BEGIN
	//=============================================================================
	// SIEMENS AG
	// (c)Copyright 2023
	//-----------------------------------------------------------------------------
	// Library:       LKinCtrl
	// Tested with:   S7-1518TF-4 PN/DP, FW V3.1
	// Engineering:   TIA Portal V19
	// Restrictions:  ---
	// Requirements:  S7-1500T, FW V3.0
	// Functionality: Calc rotation axis and angle from rotation matrix
	// Support: tech.team.motioncontrol@siemens.com
	// Note: Parameter comments are only available in language 'English (United States)'
	//-----------------------------------------------------------------------------
	// Change log table:
	// Version  Date       Expert in charge Changes applied
	// 01.00.00 21.09.2023 SF               First released version
	//=============================================================================
	
	#tempRadDeg := 180.0 / #PI;
	#tempRotAngle := ACOS((#rotMatrix[1, 1] + #rotMatrix[2, 2] + #rotMatrix[3, 3] - 1.0) * 0.5);
	
	IF (#tempRotAngle = 0.0) THEN
	  // No rotation
	  #tempR1 := 0.0;
	  #tempR2 := 0.0;
	  #tempR3 := 0.0;
	ELSIF (ABS(ABS(#tempRotAngle) - #PI) < #CALC_TOL) THEN
	  //Rotation vector 
	  IF (#tempRotAngle > 0.0) THEN //is + PI
	    #tempR1 := SQRT((#rotMatrix[1, 1] + 1) * 0.5);
	    #tempR2 := SQRT((#rotMatrix[2, 2] + 1) * 0.5);
	    #tempR3 := SQRT((#rotMatrix[3, 3] + 1) * 0.5);
	    #tempRotAngle := - #PI;
	  ELSE //is - PI
	    #tempR1 := -1.0 * SQRT((#rotMatrix[1, 1] + 1) * 0.5);
	    #tempR2 := -1.0 * SQRT((#rotMatrix[2, 2] + 1) * 0.5);
	    #tempR3 := -1.0 * SQRT((#rotMatrix[3, 3] + 1) * 0.5);
	    #tempRotAngle := - #PI;
	  END_IF;
	ELSE
	  // rotation vector
	  #tempResult1 := 0.5 / SIN(#tempRotAngle);
	  #tempR1 := #tempResult1 * (#rotMatrix[3, 2] - #rotMatrix[2, 3]);
	  #tempR2 := #tempResult1 * (#rotMatrix[1, 3] - #rotMatrix[3, 1]);
	  #tempR3 := #tempResult1 * (#rotMatrix[2, 1] - #rotMatrix[1, 2]);
	END_IF;
	#rotVector.x := #tempR1;
	#rotVector.y := #tempR2;
	#rotVector.z := #tempR3;
	#rotAngle := #tempRotAngle * #tempRadDeg;
	
END_FUNCTION

FUNCTION "LKinCtrl_RotVecToRotMatrix" : Void
TITLE = LKinCtrl_RotVecToRotMatrix
{ S7_Optimized_Access := 'TRUE' }
AUTHOR : 'handling.team.automation@siemens.com'
FAMILY : LKinCtrl
VERSION : 5.0
//Calculate rotation matrix from rotation vector and angle
   VAR_INPUT 
      rotVector : "LKinCtrl_typeCOff3DPoint";   // Rotation vector
      rotAngle : LReal;   // Rotation angle
   END_VAR

   VAR_OUTPUT 
      rotMatrix : Array[1..3, 1..3] of LReal;   // Rotation matrix
   END_VAR

   VAR_TEMP 
      tempIndex1 : Int;
      tempIndex2 : Int;
      tempRotMatrix : Array[1..3, 1..3] of LReal;
      tempRotAxis : "LKinCtrl_typeCOff3DPoint";
      tempRotAngle : LReal;
      tempDegRad : LReal;
   END_VAR

   VAR CONSTANT 
      PI : LReal := 3.14159265358979;   // Pi
      CALC_TOL : LReal := 0.001;   // Tolerance
   END_VAR


BEGIN
	//=============================================================================
	// SIEMENS AG
	// (c)Copyright 2023
	//-----------------------------------------------------------------------------
	// Library:       LKinCtrl
	// Tested with:   S7-1518TF-4 PN/DP, FW V3.1
	// Engineering:   TIA Portal V19
	// Restrictions:  ---
	// Requirements:  S7-1500T, FW V3.0
	// Functionality: Calc rotation matrix from rotation axis and angle
	// Support: tech.team.motioncontrol@siemens.com
	// Note: Parameter comments are only available in language 'English (United States)'
	//-----------------------------------------------------------------------------
	// Change log table:
	// Version  Date       Expert in charge Changes applied
	// 01.00.00 21.09.2023 SF               First released version
	//=============================================================================
	
	//init values
	FOR #tempIndex1 := 1 TO 3 DO
	  FOR #tempIndex2 := 1 TO 3 DO
	    #tempRotMatrix[#tempIndex1, #tempIndex2] := 0.0;
	  END_FOR;
	END_FOR;
	
	//create unit vec
	#tempRotAxis := "LKinCtrl_VecUnit"(#rotVector);
	//deg to rad for rot angle
	#tempDegRad := #PI / 180.0;
	#tempRotAngle := #rotAngle * #tempDegRad;
	//no rotation?
	IF (#tempRotAxis.x = 0.0 AND #tempRotAxis.y = 0.0 AND #tempRotAxis.z = 0.0) OR #tempRotAngle = 0.0 THEN
	  #rotMatrix[1, 1] := 1.0;
	  #rotMatrix[2, 2] := 1.0;
	  #rotMatrix[3, 3] := 1.0;
	  RETURN;
	END_IF;
	
	//create rotation matrix
	#rotMatrix[1, 1] := #tempRotAxis.x * #tempRotAxis.x * (1.0 - COS(#tempRotAngle)) + COS(#tempRotAngle);
	#rotMatrix[1, 2] := #tempRotAxis.x * #tempRotAxis.y * (1.0 - COS(#tempRotAngle)) - #tempRotAxis.z * SIN(#tempRotAngle);
	#rotMatrix[1, 3] := #tempRotAxis.x * #tempRotAxis.z * (1.0 - COS(#tempRotAngle)) + #tempRotAxis.y * SIN(#tempRotAngle);
	
	#rotMatrix[2, 1] := #tempRotAxis.y * #tempRotAxis.x * (1.0 - COS(#tempRotAngle)) + #tempRotAxis.z * SIN(#tempRotAngle);
	#rotMatrix[2, 2] := #tempRotAxis.y * #tempRotAxis.y * (1.0 - COS(#tempRotAngle)) + COS(#tempRotAngle);
	#rotMatrix[2, 3] := #tempRotAxis.y * #tempRotAxis.z * (1.0 - COS(#tempRotAngle)) - #tempRotAxis.x * SIN(#tempRotAngle);
	
	#rotMatrix[3, 1] := #tempRotAxis.z * #tempRotAxis.x * (1.0 - COS(#tempRotAngle)) - #tempRotAxis.y * SIN(#tempRotAngle);
	#rotMatrix[3, 2] := #tempRotAxis.z * #tempRotAxis.y * (1.0 - COS(#tempRotAngle)) + #tempRotAxis.x * SIN(#tempRotAngle);
	#rotMatrix[3, 3] := #tempRotAxis.z * #tempRotAxis.z * (1.0 - COS(#tempRotAngle)) + COS(#tempRotAngle);
	
	
	
END_FUNCTION

FUNCTION "LKinCtrl_GetDistanceToPrevious" : Word
TITLE = LKinCtrl_GetDistanceToPrevious
{ S7_Optimized_Access := 'TRUE' }
AUTHOR : 'handling.team.automation@siemens.com'
FAMILY : LKinCtrl
VERSION : 5.0
   VAR_IN_OUT 
      cmdPar : "LKinCtrl_typePnPLinCmdSeqParameter";   // Parameters of points
      axesGroup {InstructionName := 'TO_Kinematics'; LibVersion := '9.0'} : TO_Kinematics;   // Reference to axes group
   END_VAR

   VAR_TEMP 
      tempPrevPoint : "LKinCtrl_typePnPLinPointParameter" := ((), [()], (), (), [-1.0], ((), (), ((), (), (), (), (), ()), ((), (), (), (), (), ())), (), ((), (), (), ()), (), ());
      tempWord : Word;
   END_VAR

   VAR CONSTANT 
      STATUS_NO_ERR : Word := 16#0000;   // No error
      ERR_GET_DIST : Word := 16#8000;   // Error - Get linear distance
   END_VAR


BEGIN
	//=============================================================================
	// SIEMENS AG
	// (c)Copyright 2023
	//-----------------------------------------------------------------------------
	// Library:       LKinCtrl
	// Tested with:   S7-1518TF-4 PN/DP, FW V3.1
	// Engineering:   TIA Portal V19
	// Restrictions:  ---
	// Requirements:  S7-1500T, FW V3.0
	// Functionality: This block is filling the distance-parameter for a command sequence
	//                (Usage for LKinCtrl_MC_MovePickAndPlace...)
	// Support: tech.team.motioncontrol@siemens.com
	// Note: Parameter comments are only available in language 'English (United States)'
	//-----------------------------------------------------------------------------
	// Change log table:
	// Version  Date       Expert in charge Changes applied
	// 01.00.00 21.09.2023 SF               First released version
	//=============================================================================
	
	#LKinCtrl_GetDistanceToPrevious := #STATUS_NO_ERR;
	
	//Target point
	IF (#cmdPar.target.usePoint = TRUE) THEN
	  IF (#cmdPar.preTarget.usePoint = TRUE) THEN
	    #tempPrevPoint := #cmdPar.preTarget;
	  ELSIF (#cmdPar.intermediate.usePoint = TRUE) THEN
	    #tempPrevPoint := #cmdPar.intermediate;
	  ELSIF (#cmdPar.postStart.usePoint = TRUE) THEN
	    #tempPrevPoint := #cmdPar.postStart;
	  ELSE
	    #tempPrevPoint := #cmdPar.start;
	  END_IF;
	  #tempWord := "LKinCtrl_CalcLinearDistance"(previous := #tempPrevPoint,
	                                             actual := #cmdPar.target,
	                                             axesGroup := #axesGroup);
	  IF (#tempWord.%X15 = TRUE) THEN
	    #LKinCtrl_GetDistanceToPrevious := #ERR_GET_DIST;
	    RETURN;
	  END_IF;
	END_IF;
	
	//Pretarget
	IF (#cmdPar.preTarget.usePoint = TRUE) THEN
	  IF (#cmdPar.intermediate.usePoint = TRUE) THEN
	    #tempPrevPoint := #cmdPar.intermediate;
	  ELSIF (#cmdPar.postStart.usePoint = TRUE) THEN
	    #tempPrevPoint := #cmdPar.postStart;
	  ELSE
	    #tempPrevPoint := #cmdPar.start;
	  END_IF;
	  #tempWord := "LKinCtrl_CalcLinearDistance"(previous := #tempPrevPoint,
	                                             actual := #cmdPar.preTarget,
	                                             axesGroup := #axesGroup);
	  IF (#tempWord.%X15 = TRUE) THEN
	    #LKinCtrl_GetDistanceToPrevious := #ERR_GET_DIST;
	    RETURN;
	  END_IF;
	END_IF;
	
	//Intermediate
	IF (#cmdPar.intermediate.usePoint = TRUE) THEN
	  IF (#cmdPar.postStart.usePoint = TRUE) THEN
	    #tempPrevPoint := #cmdPar.postStart;
	  ELSE
	    #tempPrevPoint := #cmdPar.start;
	  END_IF;
	  #tempWord := "LKinCtrl_CalcLinearDistance"(previous := #tempPrevPoint,
	                                             actual := #cmdPar.intermediate,
	                                             axesGroup := #axesGroup);
	  IF (#tempWord.%X15 = TRUE) THEN
	    #LKinCtrl_GetDistanceToPrevious := #ERR_GET_DIST;
	    RETURN;
	  END_IF;
	END_IF;
	
	//PostStart
	IF (#cmdPar.postStart.usePoint = TRUE) THEN
	  #tempPrevPoint := #cmdPar.start;
	  #tempWord := "LKinCtrl_CalcLinearDistance"(previous := #tempPrevPoint,
	                                             actual := #cmdPar.postStart,
	                                             axesGroup := #axesGroup);
	  IF (#tempWord.%X15 = TRUE) THEN
	    #LKinCtrl_GetDistanceToPrevious := #ERR_GET_DIST;
	    RETURN;
	  END_IF;
	END_IF;
	
END_FUNCTION

FUNCTION "LKinCtrl_CalcLinearDistance" : Word
TITLE = LKinCtrl_CalcLinearDistance
{ S7_Optimized_Access := 'TRUE' }
AUTHOR : 'handling.team.automation@siemens.com'
FAMILY : LKinCtrl
VERSION : 5.0
//Calculation of the linear distance between two points (WCS or OCS)
   VAR_INPUT 
      previous : "LKinCtrl_typePnPLinPointParameter";   // Previous point info
   END_VAR

   VAR_IN_OUT 
      actual : "LKinCtrl_typePnPLinPointParameter";   // Actual point info
      axesGroup {InstructionName := 'TO_Kinematics'; LibVersion := '9.0'} : TO_Kinematics;   // Reference to axes group
   END_VAR

   VAR_TEMP 
      tempPrevPointWCS : Array[1..6] of LReal;
      tempPrevPointOCS : Array[1..6] of LReal;
      tempActPointWCS : Array[1..6] of LReal;
      tempActPointOCS : Array[1..6] of LReal;
      tempPrevPointWCS3D : "LKinCtrl_typeCOff3DPoint";
      tempActPointWCS3D : "LKinCtrl_typeCOff3DPoint";
   END_VAR

   VAR CONSTANT 
      STATUS_NO_ERR : Word := 16#0000;   // No error
      ERR_POINT_NOT_USED : Word := 16#8000;   // Error - Point is not used
   END_VAR


BEGIN
	//=============================================================================
	// SIEMENS AG
	// (c)Copyright 2023
	//-----------------------------------------------------------------------------
	// Library:       LKinCtrl
	// Tested with:   S7-1518TF-4 PN/DP, FW V3.1
	// Engineering:   TIA Portal V19
	// Restrictions:  ---
	// Requirements:  S7-1500T, FW V3.0
	// Functionality: This block is calculating the linear distance between two points (WCS or OCS)
	//                (Usage for LKinCtrl_MC_MovePickAndPlace...)
	// Support: tech.team.motioncontrol@siemens.com
	// Note: Parameter comments are only available in language 'English (United States)'
	//-----------------------------------------------------------------------------
	// Change log table:
	// Version  Date       Expert in charge Changes applied
	// 01.00.00 21.09.2023 SF               First released version
	//=============================================================================
	
	#LKinCtrl_CalcLinearDistance := #STATUS_NO_ERR;
	
	REGION CHECK_INPUT
	  IF (#actual.usePoint = FALSE) THEN
	    #LKinCtrl_CalcLinearDistance := #ERR_POINT_NOT_USED;
	    RETURN;
	  END_IF;
	  IF (#previous.usePoint = FALSE) THEN
	    //input -1 as distance
	    #actual.distanceToPrevious := -1.0;
	    RETURN;
	  END_IF;
	END_REGION
	
	REGION FRAME_TO_WCS
	  //Start in OCS?
	  IF (#previous.coordSystem >= "CS_OCS1") AND (#previous.coordSystem <= "CS_OCS3") THEN
	    #tempPrevPointOCS := #previous.position;
	    IF (#previous.tracking.active = TRUE) THEN
	      //in tracking - add object position
	      #tempPrevPointOCS[1] += #previous.tracking.objectPosition.x;
	    END_IF;
	    //Frame to WCS
	    "LKinCtrl_OcsToWcs"(ocsX := #axesGroup.StatusOcsFrame[#previous.coordSystem].x,
	                        ocsY := #axesGroup.StatusOcsFrame[#previous.coordSystem].y,
	                        ocsZ := #axesGroup.StatusOcsFrame[#previous.coordSystem].z,
	                        ocsA := #axesGroup.StatusOcsFrame[#previous.coordSystem].a,
	                        ocsB := #axesGroup.StatusOcsFrame[#previous.coordSystem].b,
	                        ocsC := #axesGroup.StatusOcsFrame[#previous.coordSystem].c,
	                        pointXOcs := #tempPrevPointOCS[1],
	                        pointYOcs := #tempPrevPointOCS[2],
	                        pointZOcs := #tempPrevPointOCS[3],
	                        pointAOcs := #tempPrevPointOCS[4],
	                        pointBOcs := #tempPrevPointOCS[5],
	                        pointCOcs := #tempPrevPointOCS[6],
	                        pointXWcs => #tempPrevPointWCS[1],
	                        pointYWcs => #tempPrevPointWCS[2],
	                        pointZWcs => #tempPrevPointWCS[3],
	                        pointAWcs => #tempPrevPointWCS[4],
	                        pointBWcs => #tempPrevPointWCS[5],
	                        pointCWcs => #tempPrevPointWCS[6]);
	  ELSE
	    #tempPrevPointWCS := #previous.position;
	  END_IF;
	  
	  //Actual in OCS?
	  IF (#actual.coordSystem >= "CS_OCS1") AND (#actual.coordSystem <= "CS_OCS3") THEN
	    #tempActPointOCS := #actual.position;
	    IF (#actual.tracking.active = TRUE) THEN
	      //in tracking - add object position
	      #tempActPointOCS[1] += #actual.tracking.objectPosition.x;
	    END_IF;
	    //Frame to WCS
	    "LKinCtrl_OcsToWcs"(ocsX := #axesGroup.StatusOcsFrame[#actual.coordSystem].x,
	                        ocsY := #axesGroup.StatusOcsFrame[#actual.coordSystem].y,
	                        ocsZ := #axesGroup.StatusOcsFrame[#actual.coordSystem].z,
	                        ocsA := #axesGroup.StatusOcsFrame[#actual.coordSystem].a,
	                        ocsB := #axesGroup.StatusOcsFrame[#actual.coordSystem].b,
	                        ocsC := #axesGroup.StatusOcsFrame[#actual.coordSystem].c,
	                        pointXOcs := #tempActPointOCS[1],
	                        pointYOcs := #tempActPointOCS[2],
	                        pointZOcs := #tempActPointOCS[3],
	                        pointAOcs := #tempActPointOCS[4],
	                        pointBOcs := #tempActPointOCS[5],
	                        pointCOcs := #tempActPointOCS[6],
	                        pointXWcs => #tempActPointWCS[1],
	                        pointYWcs => #tempActPointWCS[2],
	                        pointZWcs => #tempActPointWCS[3],
	                        pointAWcs => #tempActPointWCS[4],
	                        pointBWcs => #tempActPointWCS[5],
	                        pointCWcs => #tempActPointWCS[6]);
	  ELSE
	    #tempActPointWCS := #actual.position;
	  END_IF;
	END_REGION
	
	REGION CALC_DISTANCE
	  #tempPrevPointWCS3D.x := #tempPrevPointWCS[1];
	  #tempPrevPointWCS3D.y := #tempPrevPointWCS[2];
	  #tempPrevPointWCS3D.z := #tempPrevPointWCS[3];
	  
	  #tempActPointWCS3D.x := #tempActPointWCS[1];
	  #tempActPointWCS3D.y := #tempActPointWCS[2];
	  #tempActPointWCS3D.z := #tempActPointWCS[3];
	  
	  #actual.distanceToPrevious := "LKinCtrl_VecAbs"("LKinCtrl_VecSub"(vIn1 := #tempActPointWCS3D, vIn2 := #tempPrevPointWCS3D));
	END_REGION
	
END_FUNCTION

FUNCTION "LKinCtrl_ParametrizeLinAbsInstance" : Void
TITLE = LKinCtrl_ParametrizeLinAbsInstance
{ S7_Optimized_Access := 'TRUE' }
AUTHOR : 'handling.team.automation@siemens.com'
FAMILY : LKinCtrl
VERSION : 5.0
//Parametrizie MC_MoveLinearAbsolute instance
   VAR_INPUT 
      cmdPar : "LKinCtrl_typePnPLinPointParameter";   // Command parameter
   END_VAR

   VAR_IN_OUT 
      cmdInstance {InstructionName := 'MC_MOVELINEARABSOLUTE'; LibVersion := '9.0'} : MC_MOVELINEARABSOLUTE;   // MC_MoveLinearAbsolute Instance
   END_VAR


BEGIN
	//=============================================================================
	// SIEMENS AG
	// (c)Copyright 2023
	//-----------------------------------------------------------------------------
	// Library:       LKinCtrl
	// Tested with:   S7-1518TF-4 PN/DP, FW V3.1
	// Engineering:   TIA Portal V19
	// Restrictions:  ---
	// Requirements:  S7-1500T, FW V3.0
	// Functionality: Parametrize MC_MoveLinearAbsolute instance
	//                (Usage for LKinCtrl_MC_MovePickAndPlace...)
	// Support: tech.team.motioncontrol@siemens.com
	// Note: Parameter comments are only available in language 'English (United States)'
	//-----------------------------------------------------------------------------
	// Change log table:
	// Version  Date       Expert in charge Changes applied
	// 01.00.00 21.09.2023 SF               First released version
	//=============================================================================
	
	//Set values
	#cmdInstance.Position := #cmdPar.position;
	#cmdInstance.CoordSystem := #cmdPar.coordSystem;
	#cmdInstance.Velocity := #cmdPar.pathDynamics.velocity;
	#cmdInstance.Acceleration := #cmdPar.pathDynamics.acceleration;
	#cmdInstance.Deceleration := #cmdPar.pathDynamics.deceleration;
	#cmdInstance.Jerk := #cmdPar.pathDynamics.jerk;
	#cmdInstance.DynamicAdaption := #cmdPar.dynamicAdaption;
	#cmdInstance.DirectionA := #cmdPar.directionA;
	#cmdInstance.BufferMode := #cmdPar.bufferMode;
	#cmdInstance.TransitionParameter := #cmdPar.transitionParameter;
	
	
END_FUNCTION

FUNCTION "LKinCtrl_InitTODataRestore" : Void
TITLE = LKinCtrl_InitTODataRestore
{ S7_Optimized_Access := 'TRUE' }
AUTHOR : 'handling.team.automation@siemens.com'
FAMILY : LKinCtrl
VERSION : 5.0
//Restore specific TO data
   VAR_INPUT 
      initTOData : "LKinCtrl_typePnPInitTOData";   // Inital TO data
   END_VAR

   VAR_IN_OUT 
      axesGroup {InstructionName := 'TO_Kinematics'; LibVersion := '9.0'} : TO_Kinematics;   // Reference to axes group
   END_VAR


BEGIN
	//=============================================================================
	// SIEMENS AG
	// (c)Copyright 2023
	//-----------------------------------------------------------------------------
	// Library:       LKinCtrl
	// Tested with:   S7-1518TF-4 PN/DP, FW V3.1
	// Engineering:   TIA Portal V19
	// Restrictions:  ---
	// Requirements:  S7-1500T, FW V3.0
	// Functionality: Restore specific TO data
	// Support: tech.team.motioncontrol@siemens.com
	// Note: Parameter comments are only available in language 'English (United States)'
	//-----------------------------------------------------------------------------
	// Change log table:
	// Version  Date       Expert in charge Changes applied
	// 01.00.00 21.09.2023 SF               First released version
	//=============================================================================
	
	//Blending length factor
	#axesGroup.Transition.FactorBlendingLength := #initTOData.factorBlendingLength;
	//Orientation dynamics
	#axesGroup.DynamicDefaults.Orientation.Velocity := #initTOData.orientationDefaults.velocity;
	#axesGroup.DynamicDefaults.Orientation.Acceleration := #initTOData.orientationDefaults.acceleration;
	#axesGroup.DynamicDefaults.Orientation.Deceleration := #initTOData.orientationDefaults.deceleration;
	#axesGroup.DynamicDefaults.Orientation.Jerk := #initTOData.orientationDefaults.jerk;
END_FUNCTION

FUNCTION_BLOCK "LKinCtrl_CalcRemainingDist"
TITLE = LKinCtrl_CalcRemainingDist
{ S7_Optimized_Access := 'TRUE' }
AUTHOR : 'handling.team.automation@siemens.com'
FAMILY : LKinCtrl
VERSION : 5.0
//Calculates the cartesian distance to a target point including blending. Outputs the remaining distance.
   VAR_INPUT 
      writeCmdLoggerElement : Int;   // pointer for writing logger element; incremented after writing ==> value -1 is last written element
      activeCmdLoggerElement : Int;   // pointing on active cmd in command logger; showing active element during execution ==> after SUCCESSFUL completion of path incrementation ==> value -1 is last active element
   END_VAR

   VAR_OUTPUT 
      remainingDistance { ExternalWritable := 'False'} : LReal;   // remaining distance output
   END_VAR

   VAR_IN_OUT 
      loggerElements : Array[*] of "LKinCtrl_bufferElement";   // logger array storing executed commands and specific debug data
      OCSFrames : Array[1..3] of "LKinCtrl_typeFrame";   // array of OCS frames
      userFrames : Array["LKINCTRL_CS_NO_OF_FIRST_USER_FRAME".."LKINCTRL_CS_NO_OF_LAST_USER_FRAME"] of "LKinCtrl_typeFrame";   // array of user frames
      toKinematics {InstructionName := 'TO_Kinematics'; LibVersion := '9.0'} : TO_Kinematics;   // technology object kinematics input
   END_VAR

   VAR 
      statFirstCycle { ExternalAccessible := 'False'; ExternalVisible := 'False'; ExternalWritable := 'False'} : Bool := TRUE;   // static for first cycle
      statBlendingRadius { ExternalAccessible := 'False'; ExternalVisible := 'False'; ExternalWritable := 'False'} : LReal;   // static storing for blending radius
      statRemainingDistance { ExternalAccessible := 'False'; ExternalVisible := 'False'; ExternalWritable := 'False'} : LReal;   // static storing for remaining distance
      statLowerLimitLogger { ExternalAccessible := 'False'; ExternalVisible := 'False'; ExternalWritable := 'False'} : DInt;   // lower limit of command logger
      statUpperLimitLogger { ExternalAccessible := 'False'; ExternalVisible := 'False'; ExternalWritable := 'False'} : DInt;   // upper limit of command logger
      statActiveLoggerElementOld { ExternalAccessible := 'False'; ExternalVisible := 'False'; ExternalWritable := 'False'} : DInt;   // active command logger element
   END_VAR

   VAR_TEMP 
      tempCS : DInt;   // temporary coordinate system
      tempCalc : Array[1..6] of LReal;   // temporary calculation variable
      tempPreviousTarget : Array[1..6] of LReal;   // temporary previous target
      tempCurrentTarget : Array[1..6] of LReal;   // temporary current target
      tempNextTarget : Array[1..6] of LReal;   // temporary next target
      tempDistPrevious : Array[1..6] of LReal;   // temporary distance to previous target
      tempDistNext : Array[1..6] of LReal;   // temporary distance to next target
      tempBufferMode : DInt;   // temporary buffer mode
      tempTransitionParameter : LReal;   // temporary transition paramter
      tempLengthNextCmd : LReal;   // temporary length of next command
      tempLengthPreviousCmd : LReal;   // temporary length of previous command
   END_VAR


BEGIN
	//=============================================================================
	// SIEMENS AG
	// (c)Copyright 2021
	//------------------------------------------------------------------------------------------
	// Library: LKinCtrl
	// Tested with: S7-1517T-3 PN/DP
	// Engineering: TIA Portal V16
	// Restrictions: ---
	// Requirements: S7-1500T FW 2.8
	// Functionality: LKinCtrl_CalcRemainingDist
	// The FB calculates the cartesian distance to a target point and outputs the remaining distance to it
	//
	// Support: tech.team.motioncontrol@siemens.com
	// Note: Parameter comments are only available in language 'English (United States)'
	//------------------------------------------------------------------------------------------
	// Change log table:
	// Version    Date          Expert in charge    Changes applied
	// 01.00.00   19.05.2021    FR                  First released version
	//===========================================================================================
	
	// Init output
	#remainingDistance := 0;
	
	IF #statFirstCycle THEN
	    // Get logger limits
	    #statLowerLimitLogger := LOWER_BOUND(ARR := #loggerElements, DIM := 1);
	    #statUpperLimitLogger := UPPER_BOUND(ARR := #loggerElements, DIM := 1);
	    
	    // Check limits
	    IF #statLowerLimitLogger = #statUpperLimitLogger THEN
	        RETURN;
	    END_IF;
	    
	    #statActiveLoggerElementOld := #statLowerLimitLogger - 1; // Make sure old var is different to actual
	    #statFirstCycle := FALSE;
	END_IF;
	
	
	REGION CALCULATE_BLENDING_RADIUS
	    // Check if new command is active
	    IF #activeCmdLoggerElement <> #statActiveLoggerElementOld THEN
	        // ------------------
	        // Store old var
	        // ------------------
	        #statActiveLoggerElementOld := #activeCmdLoggerElement;
	        
	        // ------------------
	        // Get current target position
	        // ------------------
	        #tempCurrentTarget[1] := #loggerElements[#activeCmdLoggerElement].position[1];  //x coordinate
	        #tempCurrentTarget[2] := #loggerElements[#activeCmdLoggerElement].position[2];  //y coordinate
	        #tempCurrentTarget[3] := #loggerElements[#activeCmdLoggerElement].position[3];  //z coordinate
	        
	        // ------------------
	        // Get coord system
	        // ------------------
	        #tempCS := DINT_TO_INT(#loggerElements[#activeCmdLoggerElement].coordinateSystem);
	        // Only calculate if not in MCS
	        IF #tempCS = "CS_MCS" THEN
	            RETURN;
	        END_IF;
	        
	        // ------------------
	        // Get next target position
	        // ------------------
	        IF #activeCmdLoggerElement <> #statUpperLimitLogger THEN
	            IF #activeCmdLoggerElement + 1 <> #writeCmdLoggerElement THEN
	                #tempBufferMode := #loggerElements[#activeCmdLoggerElement + 1].bufferMode;
	                #tempTransitionParameter := #loggerElements[#activeCmdLoggerElement + 1].transitionParameter;
	                #tempNextTarget[1] := #loggerElements[#activeCmdLoggerElement + 1].position[1];
	                #tempNextTarget[2] := #loggerElements[#activeCmdLoggerElement + 1].position[2];
	                #tempNextTarget[3] := #loggerElements[#activeCmdLoggerElement + 1].position[3];
	                "LKinCtrl_FrameTrans"(coordSystem := #tempCS,
	                                      coordSystemOld := #loggerElements[#activeCmdLoggerElement + 1].coordinateSystem,
	                                      OCSFrames := #OCSFrames,
	                                      userFrames := #userFrames,
	                                      position := #tempNextTarget);
	            END_IF;
	        ELSE
	            IF #writeCmdLoggerElement <> 1 THEN
	                #tempBufferMode := #loggerElements[1].bufferMode;
	                #tempTransitionParameter := #loggerElements[1].transitionParameter;
	                #tempNextTarget[1] := #loggerElements[1].position[1];
	                #tempNextTarget[2] := #loggerElements[1].position[2];
	                #tempNextTarget[3] := #loggerElements[1].position[3];
	                "LKinCtrl_FrameTrans"(coordSystem := #tempCS,
	                                      coordSystemOld := #loggerElements[1].coordinateSystem,
	                                      OCSFrames := #OCSFrames,
	                                      userFrames := #userFrames,
	                                      position := #tempNextTarget);
	            END_IF;
	        END_IF;
	        
	        // ------------------
	        // Get previous target position
	        // ------------------
	        IF #activeCmdLoggerElement <> 1 THEN
	            IF #activeCmdLoggerElement - 1 <> #writeCmdLoggerElement THEN
	                #tempPreviousTarget[1] := #loggerElements[#activeCmdLoggerElement - 1].position[1];
	                #tempPreviousTarget[2] := #loggerElements[#activeCmdLoggerElement - 1].position[2];
	                #tempPreviousTarget[3] := #loggerElements[#activeCmdLoggerElement - 1].position[3];
	                "LKinCtrl_FrameTrans"(coordSystem := #tempCS,
	                                      coordSystemOld := #loggerElements[#activeCmdLoggerElement - 1].coordinateSystem,
	                                      OCSFrames := #OCSFrames,
	                                      userFrames := #userFrames,
	                                      position := #tempPreviousTarget);
	            END_IF;
	        ELSE
	            IF #statUpperLimitLogger <> #writeCmdLoggerElement THEN
	                #tempPreviousTarget[1] := #loggerElements[#statUpperLimitLogger].position[1];
	                #tempPreviousTarget[2] := #loggerElements[#statUpperLimitLogger].position[2];
	                #tempPreviousTarget[3] := #loggerElements[#statUpperLimitLogger].position[3];
	                "LKinCtrl_FrameTrans"(coordSystem := #tempCS,
	                                      coordSystemOld := #loggerElements[1].coordinateSystem,
	                                      OCSFrames := #OCSFrames,
	                                      userFrames := #userFrames,
	                                      position := #tempPreviousTarget);
	            END_IF;
	        END_IF;
	        
	        // ------------------
	        // Calc length of first command 
	        // ------------------
	        #tempDistPrevious[1] := #tempCurrentTarget[1] - #tempPreviousTarget[1];
	        #tempDistPrevious[2] := #tempCurrentTarget[2] - #tempPreviousTarget[2];
	        #tempDistPrevious[3] := #tempCurrentTarget[3] - #tempPreviousTarget[3];
	        
	        // Calculate length of vector (last to actual)
	        #tempLengthPreviousCmd := SQRT(#tempDistPrevious[1] * #tempDistPrevious[1] + #tempDistPrevious[2] * #tempDistPrevious[2] + #tempDistPrevious[3] * #tempDistPrevious[3]);
	        
	        
	        // ------------------
	        // Calc length of second command
	        // ------------------
	        #tempDistNext[1] := #tempNextTarget[1] - #tempCurrentTarget[1];
	        #tempDistNext[2] := #tempNextTarget[2] - #tempCurrentTarget[2];
	        #tempDistNext[3] := #tempNextTarget[3] - #tempCurrentTarget[3];
	        
	        // Calculate length of vector (actual to next)
	        #tempLengthNextCmd := SQRT(#tempDistNext[1] * #tempDistNext[1] + #tempDistNext[2] * #tempDistNext[2] + #tempDistNext[3] * #tempDistNext[3]);
	        
	        // ------------------
	        // Check blending settings
	        // ------------------
	        IF (#tempBufferMode = "BM_BLENDING_LOW" OR #tempBufferMode = "BM_BLENDING_HIGH") AND #tempTransitionParameter <> 0.0 THEN
	            // Check which command is shorter distance
	            IF #tempTransitionParameter < 0.0 THEN // Transition parameter 
	                // Check which command is shorter     //Last target to current              //Current target to next
	                #statBlendingRadius := MIN_LREAL(IN1 := #tempLengthPreviousCmd / 2.0, IN2 := #tempLengthNextCmd / 2.0);
	            ELSE
	                // Check which setting is the shortest
	                #statBlendingRadius := MIN_LREAL(IN1 := #tempLengthPreviousCmd / 2.0, IN2 := #tempLengthNextCmd / 2.0, IN3 := #tempTransitionParameter);
	            END_IF;
	        ELSE
	            #statBlendingRadius := 0; // Blending is deactivated at command
	        END_IF;
	    ELSE
	        ; // Blending radius is already calculated -> Nothing to do
	    END_IF;
	END_REGION
	
	REGION CALC_REMAINING_DISTANCE
	    // Substract kinematics position
	    IF #tempCS = "CS_WCS" THEN
	        #tempCalc[1] := #tempCurrentTarget[1] - #toKinematics.TcpInWcs.x.Position;
	        #tempCalc[2] := #tempCurrentTarget[2] - #toKinematics.TcpInWcs.y.Position;
	        #tempCalc[3] := #tempCurrentTarget[3] - #toKinematics.TcpInWcs.z.Position;
	    ELSE
	        #tempCalc[1] := #tempCurrentTarget[1] - #toKinematics.TcpInOcs[#tempCS].x.Position;
	        #tempCalc[2] := #tempCurrentTarget[2] - #toKinematics.TcpInOcs[#tempCS].y.Position;
	        #tempCalc[3] := #tempCurrentTarget[3] - #toKinematics.TcpInOcs[#tempCS].z.Position;
	    END_IF;
	    
	    // Remaining distance of current command
	    #statRemainingDistance := SQRT(#tempCalc[1] * #tempCalc[1] + #tempCalc[2] * #tempCalc[2] + #tempCalc[3] * #tempCalc[3]);
	END_REGION CALC_REMAINING_DISTANCE
	
	REGION SUBSTARCT_BLENDING
	    // Calculate remaining distance
	    #statRemainingDistance := #statRemainingDistance - #statBlendingRadius;
	    IF #statRemainingDistance < 0.0 THEN // Avoid negative values
	        #statRemainingDistance := 0.0;
	    END_IF;
	    
	    // Assign output
	    #remainingDistance := #statRemainingDistance;
	END_REGION SUBSTARCT_BLENDING
	
	
	
END_FUNCTION_BLOCK

FUNCTION "LKinCtrl_SetOrientationDyn" : Bool
TITLE = LKinCtrl_SetOrientationDyn
{ S7_Optimized_Access := 'TRUE' }
AUTHOR : 'handling.team.automation@siemens.com'
FAMILY : LKinCtrl
VERSION : 5.0
//Set orientation dynamics in TO Kinematics defaults
   VAR_INPUT 
      orientationDynamics : "LKinCtrl_typePathDynamics";   // Orientation dynamics to be set
   END_VAR

   VAR_IN_OUT 
      orientationDefaults {InstructionName := 'TO_Struct_Kinematics_OrientationDynamics'; LibVersion := '9.0'} : TO_Struct_Kinematics_OrientationDynamics;   // Orientation dynamic defaults of TO Kinematics
   END_VAR


BEGIN
	//==========================================================================================
	// SIEMENS AG
	// (c)Copyright 2022 All Rights Reserved
	//------------------------------------------------------------------------------------------
	// Library: LKinCtrl
	// Tested with: S7-1517T-3 PN/DP
	// Engineering: TIA Portal V16
	// Restrictions: ---
	// Requirements: S7-1500T FW 2.8
	// Functionality: LKinCtrl_SetOrientationDyn
	// The FC changes the default orientation dynamics of a given TO Kinematics
	//
	// Support: tech.team.motioncontrol@siemens.com
	// Note: Parameter comments are only available in language 'English (United States)'
	//------------------------------------------------------------------------------------------
	// Change log table:
	// Version    Date          Expert in charge    Changes applied
	// 01.00.00   04.04.2022    FR                  First released version
	//===========================================================================================
	
	// Set return value to false by default
	#LKinCtrl_SetOrientationDyn := FALSE;
	
	// Velocity
	IF #orientationDynamics.velocity > 0.0 THEN
	    #orientationDefaults.Velocity := #orientationDynamics.velocity;
	    #LKinCtrl_SetOrientationDyn := TRUE;
	END_IF;
	
	// Acceleration
	IF #orientationDynamics.acceleration > 0.0 THEN
	    #orientationDefaults.Acceleration := #orientationDynamics.acceleration;
	    #LKinCtrl_SetOrientationDyn := TRUE;
	END_IF;
	
	// Deceleration
	IF #orientationDynamics.deceleration > 0.0 THEN
	    #orientationDefaults.Deceleration := #orientationDynamics.deceleration;
	    #LKinCtrl_SetOrientationDyn := TRUE;
	END_IF;
	
	// Jerk
	IF #orientationDynamics.jerk >= 0.0 THEN
	    #orientationDefaults.Jerk := #orientationDynamics.jerk;
	    #LKinCtrl_SetOrientationDyn := TRUE;
	END_IF;
	
	
END_FUNCTION

FUNCTION "LKinCtrl_CartesianStopDistance" : Word
TITLE = LKinCtrl_CartesianStopDistance
{ S7_Optimized_Access := 'TRUE' }
AUTHOR : 'handling.team.automation@siemens.com'
FAMILY : LKinCtrl
VERSION : 5.0
//Calcualte cartesian stop distance
   VAR_INPUT 
      velX : LReal;   // WCS velocity X
      velY : LReal;   // WCS velocity Y
      velZ : LReal;   // WCS velocity Z
      accX : LReal;   // WCS acceleration X
      accY : LReal;   // WCS acceleration Y
      accZ : LReal;   // WCS acceleration Z
      acceleration : LReal;   // programmed path acceleration
      deceleration : LReal;   // programmed path deceleration
      jerk : LReal;   // programmed path jerk
   END_VAR

   VAR_OUTPUT 
      stopDistance : Array[1..6] of LReal;   // cartesian stop distance
   END_VAR

   VAR_TEMP 
      tempPathAccel : LReal;
      tempPathVelo : LReal;
      tempPathTangent : Array[1..3] of LReal;
      tempReturn : Word;
      tempStopDistance : LReal;
      tempStopDistanceVector : Array[1..6] of LReal;
      tempRetLCM : "LKinCtrl_typeRetProfileDist";
      tempDet1 : LReal;
      tempDet2 : LReal;
   END_VAR

   VAR CONSTANT 
      DISTANCE_FACTOR : LReal := 1.0;
      LCM_MODE_STATE_RELATED : DInt := 91;
      LCM_MODE_DIRECTION_RELATED : DInt := 173;
   END_VAR


BEGIN
	//==========================================================================================
	// SIEMENS AG
	// (c)Copyright 2021 All Rights Reserved
	//------------------------------------------------------------------------------------------
	// Library: LKinCtrl
	// Tested with: S7-1517T-3 PN/DP
	// Engineering: TIA Portal V16
	// Restrictions: ---
	// Requirements: S7-1500T FW 2.8
	// Functionality: LKinCtrl_CartesianStopDistance
	// Calc path stop vector (distance for relative positioning xyz)
	//
	// Support: tech.team.motioncontrol@siemens.com
	// Note: Parameter comments are only available in language 'English (United States)'
	//------------------------------------------------------------------------------------------
	// Change log table:
	// Version    Date          Expert in charge    Changes applied
	// 01.00.00   10.06.2021    FR                  First released version
	// 02.00.00   18.01.2022    FR                  Update to 6 axis
	//===========================================================================================
	
	//----------------------------------------------------------------------
	// Calc path stop vector (distance for relative positioning xyz)
	// Current movement must be linear
	//----------------------------------------------------------------------
	
	//predefine outputs
	#tempStopDistanceVector[1] := 0.0;
	#tempStopDistanceVector[2] := 0.0;
	#tempStopDistanceVector[3] := 0.0;
	#tempStopDistanceVector[4] := 0.0;
	#tempReturn := 16#0;
	
	// Calc path vector
	// V = T * vp -> vp = sqrt(vx^2 + vy^2 + vz^2)
	// A = T * ap + K * vp^2, suppose K = 0 (Linear tracking)
	#tempDet1 := #velX * #velX + #velY * #velY + #velZ * #velZ;
	#tempDet2 := #accX * #accX + #accY * #accY + #accZ * #accZ;
	IF #tempDet1 < 0.0 OR #tempDet2 < 0.0 THEN
	    //Plausibility error
	    #tempReturn := 16#FFFF;
	ELSE
	    //Calculate path velo and tangent
	    #tempPathVelo := SQRT(#tempDet1);
	    //Calculate path acceleration
	    #tempPathAccel := SQRT(#tempDet2);
	    //Calculate path tangent
	    IF #tempPathVelo > 0.0 THEN
	        //is path velo > 0?
	        #tempPathTangent[1] := #velX / #tempPathVelo;
	        #tempPathTangent[2] := #velY / #tempPathVelo;
	        #tempPathTangent[3] := #velZ / #tempPathVelo;
	    ELSE
	        IF #tempPathAccel > 0.0 THEN
	            //Check if acceleration is > 0?
	            #tempPathTangent[1] := #accX / #tempPathVelo;
	            #tempPathTangent[2] := #accY / #tempPathVelo;
	            #tempPathTangent[3] := #accZ / #tempPathVelo;
	        ELSE
	            //No motion
	            #tempPathTangent[1] := 0.0;
	            #tempPathTangent[2] := 0.0;
	            #tempPathTangent[3] := 0.0;
	        END_IF;
	    END_IF;
	    //Calc stop distance from current path velocity to 0.0
	    #tempRetLCM := "LKinCtrl_CalcTransProfileDist"(actVelocity := #tempPathVelo,
	                                                   setVelocity := 0.0, //target velocity
	                                                   actAcceleration := #tempPathAccel,
	                                                   setAcceleration := #acceleration,
	                                                   setDeceleration := #deceleration,
	                                                   setJerk := #jerk,
	                                                   mode := #LCM_MODE_STATE_RELATED);
	    
	    
	    IF #tempRetLCM.functionResult <> 16#0 THEN
	        //error
	        #tempReturn := DINT_TO_WORD(#tempRetLCM.functionResult);
	    ELSE
	        #tempStopDistance := #tempRetLCM.dist;
	        // calculate distance vector
	        // increase accuracy by taking next interpolation step into account! (-> command usually starts in next servo cycle, depending on OB Look-Ahead)
	        #tempStopDistanceVector[1] := #DISTANCE_FACTOR * (#tempPathTangent[1] * #tempStopDistance); // + #velX * #SERVO_CYCLE_TIME + 0.5 * #accX * #SERVO_CYCLE_TIME * #SERVO_CYCLE_TIME);
	        #tempStopDistanceVector[2] := #DISTANCE_FACTOR * (#tempPathTangent[2] * #tempStopDistance); // + #velY * #SERVO_CYCLE_TIME + 0.5 * #accY * #SERVO_CYCLE_TIME * #SERVO_CYCLE_TIME);
	        #tempStopDistanceVector[3] := #DISTANCE_FACTOR * (#tempPathTangent[3] * #tempStopDistance); // + #velZ * #SERVO_CYCLE_TIME + 0.5 * #accZ * #SERVO_CYCLE_TIME * #SERVO_CYCLE_TIME);
	        #tempStopDistanceVector[4] := 0.0;
	    END_IF;
	END_IF;
	
	//Output
	//-----------------------------------------------------
	#stopDistance := #tempStopDistanceVector;
	#LKinCtrl_CartesianStopDistance := #tempReturn;
END_FUNCTION

FUNCTION "LKinCtrl_CalcTransProfileDist" : "LKinCtrl_typeRetProfileDist"
TITLE = LKinCtrl_CalcTransProfileDist
{ S7_Optimized_Access := 'TRUE' }
AUTHOR : 'handling.team.automation@siemens.com'
FAMILY : LKinCtrl
VERSION : 5.0
//Calculate distance needed to change dynamics
   VAR_INPUT 
      actVelocity : LReal;   // Start velocity
      setVelocity : LReal;   // End velocity
      actAcceleration : LReal;   // Start acceleration
      setAcceleration : LReal;   // Acceleration limit
      setDeceleration : LReal;   // Deceleration limit
      setJerk : LReal;   // Jerk limit
      mode : DInt;   // Mode
   END_VAR

   VAR_TEMP 
      tempDistPartA : "LKinCtrl_typeRetProfileDist";
      tempDistPartB : "LKinCtrl_typeRetProfileDist";
   END_VAR

   VAR CONSTANT 
      LCM_MODE_STATE_RELATED : DInt := 91;
      LCM_MODE_DIRECTION_RELATED : DInt := 173;
      LCM_ERR_WRONG_JERK_ARGUMENT : DInt := 104;
      LCM_ERR_WRONG_ACCEL_LIMIT_ARGUMENT : DInt := 101;
      LCM_ERR_WRONG_MODE_ARGUMENT : DInt := 118;
   END_VAR


BEGIN
	//================================================================================
	// SIEMENS AG
	// (c)Copyright 2016 All Rights Reserved
	//--------------------------------------------------------------------------------
	// Library:  
	// Tested with: 
	// Engineering: TIA Portal V16
	// Restrictions: -
	// Requirements: S7-1500/S7-1500T FW 2.8
	// Functionality:
	// Support: tech.team.motioncontrol@siemens.com
	// Note: Parameter comments are only available in language 'English (United States)'
	//--------------------------------------------------------------------------------
	// Change log table:
	// Version  Date        Expert in charge  Changes applied
	//
	//================================================================================
	
	REGION CHECK_INPUTS
	    // Check input values
	    IF (#setJerk < 0.0 OR #setJerk > 1.0e12) THEN
	        #LKinCtrl_CalcTransProfileDist.dist := 0.0;
	        #LKinCtrl_CalcTransProfileDist.functionResult := #LCM_ERR_WRONG_JERK_ARGUMENT;
	        RETURN;
	    ELSIF (#setAcceleration <= 0.0) THEN
	        #LKinCtrl_CalcTransProfileDist.dist := 0.0;
	        #LKinCtrl_CalcTransProfileDist.functionResult := #LCM_ERR_WRONG_ACCEL_LIMIT_ARGUMENT;
	        RETURN;
	    ELSIF (#setDeceleration <= 0.0) THEN
	        #LKinCtrl_CalcTransProfileDist.dist := 0.0;
	        #LKinCtrl_CalcTransProfileDist.functionResult := #LCM_ERR_WRONG_ACCEL_LIMIT_ARGUMENT;
	        RETURN;
	    ELSIF (#mode <> #LCM_MODE_STATE_RELATED AND #mode <> #LCM_MODE_DIRECTION_RELATED) THEN
	        #LKinCtrl_CalcTransProfileDist.dist := 0.0;
	        #LKinCtrl_CalcTransProfileDist.functionResult := #LCM_ERR_WRONG_MODE_ARGUMENT;
	        RETURN;
	    END_IF;
	END_REGION
	
	REGION CALCULATION
	    // Test if motion is reversing
	    IF ((#actVelocity > 0.0 AND #setVelocity >= 0.0) OR
	        (#actVelocity < 0.0 AND #setVelocity <= 0.0) OR
	        (#actVelocity = 0.0 AND #setVelocity = 0.0) OR
	        (#actVelocity = 0.0 AND #setVelocity > 0.0 AND #actAcceleration >= 0.0) OR
	        (#actVelocity = 0.0 AND #setVelocity < 0.0 AND #actAcceleration <= 0.0))
	    THEN
	        REGION NO_REVERSING
	            // no reversing - calc distance
	            #tempDistPartA :=
	            "LKinCtrl_SubCalcTransProfileDist"(
	                                               actVelocity := #actVelocity,
	                                               setVelocity := #setVelocity,
	                                               actAcceleration := #actAcceleration,
	                                               setAcceleration := #setAcceleration,
	                                               setDeceleration := #setDeceleration,
	                                               setJerk := #setJerk,
	                                               mode := #mode
	            );
	            #LKinCtrl_CalcTransProfileDist.dist := #tempDistPartA.dist;
	        END_REGION
	    ELSE
	        REGION REVERSING
	            // reversing - two motion parts needed
	            #tempDistPartA :=
	            "LKinCtrl_SubCalcTransProfileDist"(
	                                               actVelocity := #actVelocity,
	                                               setVelocity := 0.0, // first part - stop from act velocity
	                                               actAcceleration := #actAcceleration,
	                                               setAcceleration := #setAcceleration,
	                                               setDeceleration := #setDeceleration,
	                                               setJerk := #setJerk,
	                                               mode := #mode
	            );
	            #tempDistPartB :=
	            "LKinCtrl_SubCalcTransProfileDist"(
	                                               actVelocity := 0.0, // second part - from stop to set velocity
	                                               setVelocity := #setVelocity,
	                                               actAcceleration := 0.0,
	                                               setAcceleration := #setAcceleration,
	                                               setDeceleration := #setDeceleration,
	                                               setJerk := #setJerk,
	                                               mode := #mode
	            );
	            #LKinCtrl_CalcTransProfileDist.dist := #tempDistPartA.dist + #tempDistPartB.dist;
	        END_REGION
	    END_IF;
	    
	    REGION ERROR_EVAL
	        // detect error on calculation
	        IF (#tempDistPartA.functionResult <> 0 OR #tempDistPartB.functionResult <> 0) THEN
	            #LKinCtrl_CalcTransProfileDist.functionResult := #tempDistPartA.functionResult + #tempDistPartB.functionResult;
	            #LKinCtrl_CalcTransProfileDist.dist := 0.0;
	        END_IF;
	    END_REGION
	END_REGION
	
	
	
END_FUNCTION

FUNCTION "LKinCtrl_SubCalcTransProfileDist" : "LKinCtrl_typeRetProfileDist"
TITLE = LKinCtrl_SubCalcTransProfileDist
{ S7_Optimized_Access := 'TRUE' }
AUTHOR : 'handling.team.automation@siemens.com'
FAMILY : LKinCtrl
VERSION : 5.0
//Subfunction to LKinCtrl_CalcTransProfileDist
   VAR_INPUT 
      actVelocity : LReal;   // Start velocity
      setVelocity : LReal;   // End velocity
      actAcceleration : LReal;   // Start acceleration
      setAcceleration : LReal;   // Acceleration limit
      setDeceleration : LReal;   // Deceleration limit
      setJerk : LReal;   // Jerk limit
      mode : DInt;   // Mode
   END_VAR

   VAR_TEMP 
      tempTsum : LReal;
      tempDist : LReal;
      tempMaxAcc : LReal;
      tempMaxDec : LReal;
      tempActAcc : LReal;
      tempAcc : LReal;
      tempDec : LReal;
      tempActVel : LReal;
      tempVel : LReal;
      tempT1 : LReal;
      tempT2 : LReal;
      tempT3 : LReal;
      tempDeltaVelocity : LReal;
      tempMinJerk : LReal;
      tempSign : SInt;
      tempVelTest : LReal;
   END_VAR

   VAR CONSTANT 
      LCM_MODE_STATE_RELATED : DInt := 91;
      LCM_MODE_DIRECTION_RELATED : DInt := 173;
      LCM_ERR_JERK_OUT_OF_BOUNDS : DInt := 113;
      LCM_MINJERK_TOLERANCE : LReal := 1.0E-06;
   END_VAR


BEGIN
	//================================================================================
	// SIEMENS AG
	// (c)Copyright 2016 All Rights Reserved
	//--------------------------------------------------------------------------------
	// Library:  
	// Tested with: 
	// Engineering: TIA Portal V16
	// Restrictions: -
	// Requirements: S7-1500/S7-1500T FW 2.8
	// Functionality:
	// Support: tech.team.motioncontrol@siemens.com
	// Note: Parameter comments are only available in language 'English (United States)'
	//--------------------------------------------------------------------------------
	// Change log table:
	// Version  Date        Expert in charge  Changes applied
	//
	//================================================================================
	
	(*
	Notes on value assignment:
	The values of the initial speed or target speed are assigned so that the target speed is the greater speed in each case.
	The limits of acceleration and deceleration must also be swapped according to the mode.
	Likewise, the initial acceleration changes its sign.
	So that the distance can be returned with the correct sign, the direction of movement is noted in "tempSign".
	*)
	
	REGION GET_MOTION_DIRECTION
	    IF (#actVelocity = 0.0 AND #setVelocity = 0.0 AND #actAcceleration <= 0.0) THEN
	        #tempActVel := #actVelocity;
	        #tempVel := #setVelocity;
	        IF (#mode = #LCM_MODE_DIRECTION_RELATED) THEN
	            #tempAcc := #setAcceleration;
	            #tempDec := #setDeceleration;
	        ELSIF (#mode = #LCM_MODE_STATE_RELATED) THEN
	            #tempAcc := #setDeceleration;
	            #tempDec := #setAcceleration;
	        END_IF;
	        #tempActAcc := #actAcceleration;
	        #tempSign := 1;
	        
	    ELSIF (#actVelocity = 0.0 AND #setVelocity = 0.0 AND #actAcceleration >= 0.0) THEN
	        #tempActVel := #actVelocity;
	        #tempVel := #setVelocity;
	        #tempAcc := #setAcceleration;
	        #tempDec := #setDeceleration;
	        #tempActAcc := #actAcceleration;
	        #tempSign := 1;
	        
	    ELSIF (#actVelocity <= #setVelocity AND #actVelocity >= 0.0 AND #setVelocity >= 0.0) THEN
	        #tempActVel := #actVelocity;
	        #tempVel := #setVelocity;
	        #tempAcc := #setAcceleration;
	        #tempDec := #setDeceleration;
	        #tempActAcc := #actAcceleration;
	        #tempSign := 1;
	        
	    ELSIF (#actVelocity <= #setVelocity AND #actVelocity <= 0.0 AND #setVelocity <= 0.0) THEN
	        #tempActVel := #actVelocity;
	        #tempVel := #setVelocity;
	        IF (#mode = #LCM_MODE_DIRECTION_RELATED) THEN
	            #tempAcc := #setAcceleration;
	            #tempDec := #setDeceleration;
	        ELSIF (#mode = #LCM_MODE_STATE_RELATED) THEN
	            #tempAcc := #setDeceleration;
	            #tempDec := #setAcceleration;
	        END_IF;
	        #tempActAcc := #actAcceleration;
	        #tempSign := 1;
	        
	    ELSIF (#actVelocity >= #setVelocity AND #actVelocity >= 0.0 AND #setVelocity >= 0.0) THEN
	        #tempActVel := - #actVelocity;
	        #tempVel := - #setVelocity;
	        IF (#mode = #LCM_MODE_DIRECTION_RELATED) THEN
	            #tempAcc := #setDeceleration;
	            #tempDec := #setAcceleration;
	        ELSIF (#mode = #LCM_MODE_STATE_RELATED) THEN
	            #tempAcc := #setDeceleration;
	            #tempDec := #setAcceleration;
	        END_IF;
	        #tempActAcc := - #actAcceleration;
	        #tempSign := -1;
	        
	    ELSIF (#actVelocity >= #setVelocity AND #actVelocity <= 0.0 AND #setVelocity <= 0.0) THEN
	        #tempActVel := - #actVelocity;
	        #tempVel := - #setVelocity;
	        IF (#mode = #LCM_MODE_DIRECTION_RELATED) THEN
	            #tempAcc := #setDeceleration;
	            #tempDec := #setAcceleration;
	        ELSIF (#mode = #LCM_MODE_STATE_RELATED) THEN
	            #tempAcc := #setAcceleration;
	            #tempDec := #setDeceleration;
	        END_IF;
	        #tempActAcc := - #actAcceleration;
	        #tempSign := -1;
	        
	    END_IF;
	    #tempDeltaVelocity := #tempVel - #tempActVel;
	END_REGION
	
	REGION MOTION_CALCULATION
	    // Check if smooth or trapeziodal profile is used
	    IF (#setJerk <> 0.0) THEN
	        REGION SMOOTH_PROFILE
	            // Use smooth profile
	            // Check dynamics limits
	            IF (#tempActAcc > 0.0 AND #tempActVel < 0.0) THEN
	                #tempMinJerk := -0.5 * (#tempActAcc * #tempActAcc) / #tempActVel;
	                IF (#setJerk < #tempMinJerk * (1 - #LCM_MINJERK_TOLERANCE)) THEN
	                    #LKinCtrl_SubCalcTransProfileDist.dist := 0.0;
	                    #LKinCtrl_SubCalcTransProfileDist.functionResult := #LCM_ERR_JERK_OUT_OF_BOUNDS;
	                    RETURN;
	                    
	                END_IF;
	            END_IF;
	            IF (#tempActAcc < 0.0 AND #tempActVel > 0.0) THEN
	                #tempMinJerk := 0.5 * (#tempActAcc * #tempActAcc) / #tempActVel;
	                IF (#setJerk < #tempMinJerk * (1 - #LCM_MINJERK_TOLERANCE)) THEN
	                    #LKinCtrl_SubCalcTransProfileDist.dist := 0.0;
	                    #LKinCtrl_SubCalcTransProfileDist.functionResult := #LCM_ERR_JERK_OUT_OF_BOUNDS;
	                    RETURN;
	                    
	                END_IF;
	            END_IF;
	            #tempVelTest := (#tempActAcc * #tempActAcc) / 2.0 / #setJerk;
	            IF (#tempDeltaVelocity < #tempVelTest AND #tempActAcc > 0.0) THEN
	                // Profile 4 or 5
	                #tempTsum := #tempActAcc / #setJerk + SQRT((2.0 * (#tempActAcc * #tempActAcc) - 4.0 * #setJerk * #tempDeltaVelocity) / ((#setJerk * #setJerk)));
	                #tempT1 := #tempTsum / 2.0 + #tempActAcc / 2.0 / #setJerk;
	                #tempT2 := #tempTsum / 2.0 - #tempActAcc / 2.0 / #setJerk;
	                #tempMaxDec := #setJerk * #tempT2;  //tempMaxDec as absolute value
	                IF (#tempDec > #tempMaxDec) THEN
	                    //Profile 4
	                    #tempDist := ((#tempT2 * #tempT2 * #tempT2) - (#tempT1 * #tempT1 * #tempT1)) * #setJerk / 6.0 - #setJerk / 2.0 * #tempT1 * #tempT2 * #tempTsum + #tempTsum * (#tempActAcc / 2.0 * #tempTsum + #tempActVel);
	                    #LKinCtrl_SubCalcTransProfileDist.dist := #tempSign * #tempDist;
	                    
	                ELSE
	                    //Profile 5
	                    #tempTsum := (#tempActAcc + #tempDec) / #setJerk - #tempDeltaVelocity / #tempDec + (#tempActAcc * #tempActAcc) / 2.0 / #setJerk / #tempDec;
	                    #tempT1 := (#tempDec + #tempActAcc) / #setJerk;
	                    #tempT3 := #tempDec / #setJerk;
	                    #tempT2 := #tempTsum - #tempT1 - #tempT3;
	                    #tempDist := #setJerk / 6.0 * ((#tempT3 * #tempT3 * #tempT3) - (#tempT1 * #tempT1 * #tempT1)) - #tempDec / 2.0 * ((#tempT2 + #tempT3) * (#tempT2 + #tempT3))
	                    + #tempActVel * #tempTsum + #tempActAcc * #tempT1 * (#tempT1 / 2.0 + #tempT2 + #tempT3)
	                    - #setJerk / 2.0 * (#tempT1 * #tempT1) * (#tempT2 + #tempT3);
	                    #LKinCtrl_SubCalcTransProfileDist.dist := #tempSign * #tempDist;
	                    
	                END_IF;
	            ELSE
	                // Profile 1,2 or 3
	                IF (#tempActAcc > #tempAcc) THEN
	                    // Profile 3
	                    #tempTsum := #tempActAcc / #setJerk - (#tempActAcc * #tempActAcc) / 2.0 / #tempAcc / #setJerk + #tempDeltaVelocity / #tempAcc;
	                    #tempDist := (#tempActAcc * #tempActAcc) / (#setJerk * #setJerk) * (#tempActAcc / 3.0 - #tempAcc / 4.0 - (#tempActAcc * #tempActAcc) / 8.0 / #tempAcc)
	                    + ((#tempAcc * #tempAcc) * (#tempVel - #tempActVel) + 2.0 * #tempActAcc * #tempActVel * #tempAcc - (#tempActAcc * #tempActAcc) * #tempActVel) / 2.0 / #setJerk / #tempAcc
	                    + ((#tempVel * #tempVel) - (#tempActVel * #tempActVel)) / 2.0 / #tempAcc;
	                    #LKinCtrl_SubCalcTransProfileDist.dist := #tempSign * #tempDist;
	                    
	                ELSE
	                    // Profile 1 or 2
	                    #tempTsum := SQRT(2.0 * (#tempActAcc / #setJerk) * (#tempActAcc / #setJerk) + 4.0 / #setJerk * #tempDeltaVelocity) - #tempActAcc / #setJerk;
	                    #tempMaxAcc := (#tempActAcc + #setJerk * #tempTsum) / 2.0;
	                    IF (#tempMaxAcc <= #tempAcc) THEN
	                        // Profile 1
	                        #tempT2 := (#tempActAcc + #setJerk * #tempTsum) / (2.0 * #setJerk);
	                        #tempDist := #tempActVel * #tempTsum + 0.5 * #tempActAcc * (#tempTsum * #tempTsum) + (#setJerk / 6.0) * ((#tempTsum * #tempTsum * #tempTsum) - 2.0 * (#tempT2 * #tempT2 * #tempT2));
	                        #LKinCtrl_SubCalcTransProfileDist.dist := #tempSign * #tempDist;
	                        
	                    ELSE
	                        // Profile 2 
	                        #tempTsum := ((#tempAcc * #tempAcc) + 0.5 * (#tempActAcc * #tempActAcc) - #tempActAcc * #tempAcc + #setJerk * #tempDeltaVelocity) / (#setJerk * #tempAcc);
	                        #tempDist := #tempAcc / 2.0 / #setJerk * (#tempActVel + #tempVel) + #tempActAcc * #tempActVel / #setJerk * (#tempActAcc / 2.0 / #tempAcc - 1.0)
	                        + ((#tempVel * #tempVel) - (#tempActVel * #tempActVel)) / 2.0 / #tempAcc
	                        + ((#tempActAcc * #tempActAcc)) / (#setJerk * #setJerk) * (#tempActAcc / 3.0 - (#tempActAcc * #tempActAcc) / 8.0 / #tempAcc - #tempAcc / 4.0);
	                        #LKinCtrl_SubCalcTransProfileDist.dist := #tempSign * #tempDist;
	                        
	                    END_IF;
	                END_IF;
	            END_IF;
	        END_REGION
	    ELSE
	        REGION TRAPEZIODAL_PROFILE
	            // Use trapeziodal profile
	            #tempTsum := #tempDeltaVelocity / #tempAcc;
	            #tempDist := ((#tempVel * #tempVel) - (#tempActVel * #tempActVel)) / 2.0 / #tempAcc;
	            #LKinCtrl_SubCalcTransProfileDist.dist := #tempSign * #tempDist;
	        END_REGION
	    END_IF;
	END_REGION
	
END_FUNCTION

FUNCTION "LKinCtrl_PathDataConversion" : Word
TITLE = LKinCtrl_PathDataConversion
{ S7_Optimized_Access := 'TRUE' }
AUTHOR : 'handling.team.automation@siemens.com'
FAMILY : LKinCtrl
VERSION : 5.0
   VAR_INPUT 
      pathDataInput : Variant;   // Path data of legacy types LKinCtrl_typePathData_reduced and LKinCtrl_typePathData_advanced
   END_VAR

   VAR_OUTPUT 
      pathData : "LKinCtrl_typePathData";   // Converted path data
   END_VAR

   VAR_TEMP 
      tempRefPathDataReduced : REF_TO "LKinCtrl_typePathData_reduced";
      tempRefPathDataAdvanced : REF_TO "LKinCtrl_typePathData_advanced";
      tempRefPathData : REF_TO "LKinCtrl_typePathData";
      tempCommand : "LKinCtrl_typePathDataElement" := ((), (), (), (), (), (((), (), (), (), (), ()), ()), (((), (), (), ()), ((), (), (), ()), (), (), [-1.0], (), (), ((), (), [()]), ((), ()), (()), ((), (), [()], (), (), (), ()), ((), (), ()), (([()], (), (), ()), ([()], (), (), ()))), [((), (), ()), ((), (), ()), ((), (), ())], [((), (), (), ()), ((), (), (), ()), ((), (), (), ()), ((), (), (), ())], [6(TRUE)]);
      tempCommandReduced : "LKinCtrl_typePathDataElement_reduced" := ((), (), (), (), (((), (), (), (), (), ()), ()), (((), (), (), ()), (), (), [-1.0], ()), [((), (), ()), ((), (), ()), ((), (), ())], [((), (), (), ()), ((), (), (), ()), ((), (), (), ()), ((), (), (), ())]);
      tempIndex : DInt;
      tempIndex2 : DInt;
      tempInputPathLimit : DInt;
      tempOutputPathLimit : DInt;
   END_VAR

   VAR CONSTANT 
      NO_ERROR : Word := 16#0000;
      ERROR_INVALID_INPUT : Word := 16#8200;
      ERROR_COMMANDS_DO_NOT_FIT : Word := 16#8201;
      ERROR_INVALID_REFERENCE : Word := 16#8202;
   END_VAR


BEGIN
	//==========================================================================================
	// SIEMENS AG
	// (c)Copyright 2024 All Rights Reserved
	//------------------------------------------------------------------------------------------
	// Library: LKinCtrl
	// Tested with: S7-1517T-3 PN/DP
	// Engineering: TIA Portal V19
	// Restrictions: ---
	// Requirements: S7-1500T FW 3.1
	// Functionality: 
	// The FC converts a given legacy pathData type reduced or advanced to a regular pathData.
	// Support: tech.team.motioncontrol@siemens.com
	// Note: Parameter comments are only available in language 'English (United States)'
	//------------------------------------------------------------------------------------------
	// Change log table:
	// Version    Date          Expert in charge    Changes applied
	// 01.00.00   13.09.2024    FR                  First released version
	//===========================================================================================
	// Initialize return value
	#LKinCtrl_PathDataConversion := #NO_ERROR;
	
	// Check input type
	CASE TypeOf(#pathDataInput) OF
	  "LKinCtrl_typePathData_reduced":
	    #tempRefPathDataReduced ?= #pathDataInput;
	    
	    IF #tempRefPathDataReduced = NULL THEN
	      #LKinCtrl_PathDataConversion := #ERROR_INVALID_REFERENCE;
	      RETURN;
	    END_IF;
	    
	    #tempInputPathLimit := "LKINCTRL_NO_OF_PATHDATA_ELEMENTS_REDUCED";
	    #tempOutputPathLimit := "LKINCTRL_NO_OF_PATHDATA_ELEMENTS";
	    
	    IF #tempInputPathLimit <= #tempOutputPathLimit THEN
	      ;// Commands will fit
	    ELSE
	      // Check if there are commands after last index for regular path
	      FOR #tempIndex := #tempOutputPathLimit + 1 TO #tempInputPathLimit DO
	        IF #tempRefPathDataReduced^.commands[#tempIndex].cmdType <> -1 THEN
	          #LKinCtrl_PathDataConversion := #ERROR_COMMANDS_DO_NOT_FIT;
	          RETURN;
	        END_IF;
	      END_FOR;
	    END_IF;
	    
	    // Copy path name
	    #pathData.pathDataName := #tempRefPathDataReduced^.pathDataName;
	    
	    // Copy commands
	    FOR #tempIndex := 1 TO MIN(IN1 := #tempOutputPathLimit, IN2 := #tempInputPathLimit) DO
	      #tempCommandReduced := #tempRefPathDataReduced^.commands[#tempIndex];
	      
	      // Copy command
	      #tempCommand.cmdType := #tempCommandReduced.cmdType;
	      #tempCommand.cmdActivated := #tempCommandReduced.cmdActivated;
	      #tempCommand.cmdName := #tempCommandReduced.cmdName;
	      #tempCommand.point := #tempCommandReduced.point;
	      #tempCommand.cmdCoordinates := #tempCommandReduced.cmdCoordinates;
	      #tempCommand.cmdParameters.pathDynamics := #tempCommandReduced.cmdParameters.pathDynamics;
	      #tempCommand.cmdParameters.orientationDirection := #tempCommandReduced.cmdParameters.orientationDirection;
	      #tempCommand.cmdParameters.bufferMode := #tempCommandReduced.cmdParameters.bufferMode;
	      #tempCommand.cmdParameters.transitionParameters := #tempCommandReduced.cmdParameters.transitionParameters;
	      #tempCommand.cmdParameters.dynamicAdaption := #tempCommandReduced.cmdParameters.dynamicAdaption;
	      #tempCommand.setFlags := #tempCommandReduced.setFlags;
	      #tempCommand.valueFlags := #tempCommandReduced.valueFlags;
	      
	      // Set valid bits to true
	      FOR #tempIndex2 := 1 TO "LKINCTRL_NO_OF_VALID_BITS" DO
	        #tempCommand.parameterValid[#tempIndex2] := TRUE;
	      END_FOR;
	      
	      // Copy temp to pathData
	      #pathData.commands[#tempIndex] := #tempCommand;
	    END_FOR;
	    
	  "LKinCtrl_typePathData":
	    // Just copy input to output
	    #tempRefPathData ?= #pathDataInput;
	    
	    IF #tempRefPathData = NULL THEN
	      #LKinCtrl_PathDataConversion := #ERROR_INVALID_REFERENCE;
	      RETURN;
	    END_IF;
	    
	    #pathData := #tempRefPathData^;
	    
	  "LKinCtrl_typePathData_advanced":
	    #tempRefPathDataAdvanced ?= #pathDataInput;
	    
	    IF #tempRefPathDataAdvanced = NULL THEN
	      #LKinCtrl_PathDataConversion := #ERROR_INVALID_REFERENCE;
	      RETURN;
	    END_IF;
	    
	    #tempInputPathLimit := "LKINCTRL_NO_OF_PATHDATA_ELEMENTS_ADVANCED";
	    #tempOutputPathLimit := "LKINCTRL_NO_OF_PATHDATA_ELEMENTS";
	    
	    IF #tempInputPathLimit <= #tempOutputPathLimit THEN
	      ;// Commands will fit
	    ELSE
	      // Check if there are commands after last index for regular path
	      FOR #tempIndex := #tempOutputPathLimit + 1 TO #tempInputPathLimit DO
	        IF #tempRefPathDataAdvanced^.commands[#tempIndex].cmdType <> -1 THEN
	          #LKinCtrl_PathDataConversion := #ERROR_COMMANDS_DO_NOT_FIT;
	          RETURN;
	        END_IF;
	      END_FOR;
	    END_IF;
	    
	    // Copy path name
	    #pathData.pathDataName := #tempRefPathDataAdvanced^.pathDataName;
	    
	    // Copy commands
	    FOR #tempIndex := 1 TO MIN(IN1 := #tempOutputPathLimit, IN2 := #tempInputPathLimit) DO
	      #pathData.commands[#tempIndex] := #tempRefPathDataAdvanced^.commands[#tempIndex];
	    END_FOR;
	    
	  ELSE
	    #LKinCtrl_PathDataConversion := #ERROR_INVALID_INPUT;
	    RETURN;
	END_CASE;
	
	
	
	
	
END_FUNCTION

FUNCTION_BLOCK "LKinCtrl_GetKinematicsErrorWord"
TITLE = LKinCtrl_GetKinematicsErrorWord
{ S7_Optimized_Access := 'TRUE' }
AUTHOR : 'handling.team.automation@siemens.com'
FAMILY : LKinCtrl
VERSION : 5.0
//FB provides functionalities to reveice status information on Kinematics ErrorWord
   VAR_INPUT 
      axesGroup {InstructionName := 'TO_Kinematics'; LibVersion := '9.0'} : TO_Kinematics;   // reference to the axesGroup
   END_VAR

   VAR_OUTPUT 
      systemFault { ExternalWritable := 'False'} : Bool;   // system-internal error has occured
      configFault { ExternalWritable := 'False'} : Bool;   // one or more configuration parameters are inconsistent or invalid
      userFault { ExternalWritable := 'False'} : Bool;   // error in the user program with a Motion Control instructioc or its use
      commandNotAccepted { ExternalWritable := 'False'} : Bool;   // command cannot be accepted
      transformationFault { ExternalWritable := 'False'} : Bool;   // error in the kinematics transformation
      dynamicError { ExternalWritable := 'False'} : Bool;   // specified dynamic values are limited to permissible values
   END_VAR

   VAR 
      statFirstCycle { ExternalAccessible := 'False'; ExternalVisible := 'False'; ExternalWritable := 'False'} : Bool := TRUE;   // flag first cycle
      statErrorWordOld { ExternalAccessible := 'False'; ExternalVisible := 'False'; ExternalWritable := 'False'} : DWord;   // flag word for old errorWord
   END_VAR

   VAR_TEMP 
      tempErrorWord : DWord;
   END_VAR


BEGIN
	//==========================================================================================
	// SIEMENS AG
	// (c)Copyright 2019 All Rights Reserved
	//------------------------------------------------------------------------------------------
	// Library: LKinCtrl
	// Tested with: S7-1515T-2 PN
	// Engineering: TIA Portal V15
	// Restrictions: ---
	// Requirements: S7-1500T FW 2.5
	// Functionality: LKinCtrl_GetKinematicsErrorWord
	// The FB is splitting the error word of a technoloy object kinematic into bits.
	// Support: tech.team.motioncontrol@siemens.com
	// Note: Parameter comments are only available in language 'English (United States)'
	//------------------------------------------------------------------------------------------
	// Change log table:
	// Version    Date          Expert in charge    Changes applied
	// 01.00.00   16.08.2017    RK                  First released version
	//===========================================================================================
	
	//----------------------------------------------------------------------------------------------
	// Read errorWord
	//----------------------------------------------------------------------------------------------
	#tempErrorWord := #axesGroup.ErrorWord;
	
	//----------------------------------------------------------------------------------------------
	// Write outputs
	//----------------------------------------------------------------------------------------------
	IF #tempErrorWord <> #statErrorWordOld
	    OR #statFirstCycle
	THEN
	    #systemFault := #tempErrorWord.%X0;
	    #configFault := #tempErrorWord.%X1;
	    #userFault := #tempErrorWord.%X2;
	    #commandNotAccepted := #tempErrorWord.%X3;
	    #transformationFault := #tempErrorWord.%X4;
	    #dynamicError := #tempErrorWord.%X6;
	    
	    
	    // Set back flag
	    #statFirstCycle := False;
	ELSE
	    ; // Do nothing
	END_IF;
	
	// Copy current state of error for edge detection
	#statErrorWordOld := #tempErrorWord;
	
END_FUNCTION_BLOCK

FUNCTION_BLOCK "LKinCtrl_GetKinematicsStatusWord"
TITLE = LKinCtrl_GetKinematicsStatusWord
{ S7_Optimized_Access := 'TRUE' }
AUTHOR : 'handling.team.automation@siemens.com'
FAMILY : LKinCtrl
VERSION : 5.0
//FB provides functionalities to reveice status information on Kinematics StatusWord
   VAR_INPUT 
      axesGroup {InstructionName := 'TO_Kinematics'; LibVersion := '9.0'} : TO_Kinematics;   // reference to the axesGroup
   END_VAR

   VAR_OUTPUT 
      error { ExternalWritable := 'False'} : Bool;   // error axesGroup
      restartActive { ExternalWritable := 'False'} : Bool;   // restart of TO Kinematic active
      onlineStartValuesChanged { ExternalWritable := 'False'} : Bool;   // change of start values TO Kinematic
      controlPanelActive { ExternalWritable := 'False'} : Bool;   // control panel TO Kinematic activated
      done { ExternalWritable := 'False'} : Bool;   // no motion command active / control panel deactivated
      linearCommand { ExternalWritable := 'False'} : Bool;   // linear command active
      circularCommand { ExternalWritable := 'False'} : Bool;   // circular command active
      constantVelocity { ExternalWritable := 'False'} : Bool;   // TO Kinematic at constant velocity
      accelerating { ExternalWritable := 'False'} : Bool;   // acceleration progress active
      decelerating { ExternalWritable := 'False'} : Bool;   // deceleration progress active
      orientationMotion { ExternalWritable := 'False'} : Bool;   // orientation motion active
      stopping { ExternalWritable := 'False'} : Bool;   // MC_GroupStop is active
      interrupted { ExternalWritable := 'False'} : Bool;   // motion interrupted
      blending { ExternalWritable := 'False'} : Bool;   // no blending segment active
   END_VAR

   VAR 
      statFirstCycle { ExternalAccessible := 'False'; ExternalVisible := 'False'; ExternalWritable := 'False'} : Bool := TRUE;   // flag first cycle
      statStatusWordOld { ExternalAccessible := 'False'; ExternalVisible := 'False'; ExternalWritable := 'False'} : DWord;   // flag word for old statusWord
   END_VAR

   VAR_TEMP 
      tempStatusWord : DWord;
   END_VAR


BEGIN
	//==========================================================================================
	// SIEMENS AG
	// (c)Copyright 2019 All Rights Reserved
	//------------------------------------------------------------------------------------------
	// Library: LKinCtrl
	// Tested with: S7-1515T-2 PN
	// Engineering: TIA Portal V15
	// Restrictions: ---
	// Requirements: S7-1500T FW 2.5
	// Functionality: LKinCtrl_GetKinematicsStatusWord
	// The FB is splitting the status word of a technoloy object kinematic into bits.
	// Support: tech.team.motioncontrol@siemens.com
	// Note: Parameter comments are only available in language 'English (United States)'
	//------------------------------------------------------------------------------------------
	// Change log table:
	// Version    Date          Expert in charge    Changes applied
	// 01.00.00   16.08.2017    RK                  First released version
	//===========================================================================================
	
	//----------------------------------------------------------------------------------------------
	// Read statusword
	//----------------------------------------------------------------------------------------------
	#tempStatusWord := #axesGroup.StatusWord;
	
	//----------------------------------------------------------------------------------------------
	// Write outputs
	//----------------------------------------------------------------------------------------------
	IF #tempStatusWord <> #statStatusWordOld
	    OR #statFirstCycle
	THEN
	    #error := #tempStatusWord.%X1;
	    #restartActive := #tempStatusWord.%X2;
	    #onlineStartValuesChanged := #tempStatusWord.%X3;
	    #controlPanelActive := #tempStatusWord.%X4;
	    // #reservedBit_5 := #tempStatusWord.%X5;
	    #done := #tempStatusWord.%X6;
	    // #reservedBit_7 := #tempStatusWord.%X7;
	    #linearCommand := #tempStatusWord.%X8;
	    #circularCommand := #tempStatusWord.%X9;
	    // #polynomialCommand := #tempStatusWord.%X10;
	    // #directCommand := #tempStatusWord.%X11;
	    #constantVelocity := #tempStatusWord.%X12;
	    #accelerating := #tempStatusWord.%X13;
	    #decelerating := #tempStatusWord.%X14;
	    #orientationMotion := #tempStatusWord.%X15;
	    #stopping := #tempStatusWord.%X16;
	    #interrupted := #tempStatusWord.%X17;
	    #blending := #tempStatusWord.%X18;
	    
	    // Set back flag
	    #statFirstCycle := False;
	ELSE
	    ; // Do nothing
	END_IF;
	
	// Copy current state of status for edge detection
	#statStatusWordOld := #tempStatusWord;
	
END_FUNCTION_BLOCK

FUNCTION_BLOCK "LKinCtrl_GetKinematicsWarningWord"
TITLE = LKinCtrl_GetKinematicsWarningWord
{ S7_Optimized_Access := 'TRUE' }
AUTHOR : 'handling.team.automation@siemens.com'
FAMILY : LKinCtrl
VERSION : 5.0
//FB provides functionalities to reveice status information on Kinematics WarningWord
   VAR_INPUT 
      axesGroup {InstructionName := 'TO_Kinematics'; LibVersion := '9.0'} : TO_Kinematics;   // reference to the axesGroup
   END_VAR

   VAR_OUTPUT 
      systemFault { ExternalWritable := 'False'} : Bool;   // system-internal error has occured
      configFault { ExternalWritable := 'False'} : Bool;   // one or more configuration parameters are inconsistent or invalid
      userFault { ExternalWritable := 'False'} : Bool;   // error in the user program with a Motion Control instructioc or its use
      commandNotAccepted { ExternalWritable := 'False'} : Bool;   // command cannot be accepted
      dynamicWarning { ExternalWritable := 'False'} : Bool;   // specified dynamic values are limited to permissible values
   END_VAR

   VAR 
      statFirstCycle { ExternalAccessible := 'False'; ExternalVisible := 'False'; ExternalWritable := 'False'} : Bool := TRUE;   // flag first cycle
      statWarningWordOld { ExternalAccessible := 'False'; ExternalVisible := 'False'; ExternalWritable := 'False'} : DWord;   // flag word for old warningWord
   END_VAR

   VAR_TEMP 
      tempWarningWord : DWord;
   END_VAR


BEGIN
	//==========================================================================================
	// SIEMENS AG
	// (c)Copyright 2019 All Rights Reserved
	//------------------------------------------------------------------------------------------
	// Library: LKinCtrl
	// Tested with: S7-1515T-2 PN
	// Engineering: TIA Portal V15
	// Restrictions: ---
	// Requirements: S7-1500T FW 2.5
	// Functionality: LinCtrl_GetKinematicsWarningWord
	// The FB is splitting the warning word of a technoloy object kinematic into bits.
	// Support: tech.team.motioncontrol@siemens.com
	// Note: Parameter comments are only available in language 'English (United States)'
	//------------------------------------------------------------------------------------------
	// Change log table:
	// Version    Date          Expert in charge    Changes applied
	// 01.00.00   16.08.2017    RK                  First released version
	//===========================================================================================
	
	//----------------------------------------------------------------------------------------------
	// Read warningWord
	//----------------------------------------------------------------------------------------------
	#tempWarningWord := #axesGroup.WarningWord;
	
	//-----------------------------------------------
	//
	//
	//-----------------------------------------------
	// Write outputs
	//----------------------------------------------------------------------------------------------
	IF #tempWarningWord <> #statWarningWordOld
	    OR #statFirstCycle
	THEN
	    #systemFault := #tempWarningWord.%X0;
	    #configFault := #tempWarningWord.%X1;
	    #userFault := #tempWarningWord.%X2;
	    #commandNotAccepted := #tempWarningWord.%X3;
	    #dynamicWarning := #tempWarningWord.%X6;
	    
	    
	    // Set back flag
	    #statFirstCycle := False;
	ELSE
	    ; // Do nothing
	END_IF;
	
	// Copy current state of warning for edge detection
	#statWarningWordOld := #tempWarningWord;
	
END_FUNCTION_BLOCK

FUNCTION "LKinCtrl_FrameTransTool" : Void
TITLE = LKinCtrl_FrameTransTool
{ S7_Optimized_Access := 'TRUE' }
AUTHOR : 'handling.team.automation@siemens.com'
FAMILY : LKinCtrl
VERSION : 5.0
//Transform postion into different coordinate systems
   VAR_INPUT 
      toolResult : DInt;   // resulting tool coordinate system
      toolInitial : DInt;   // initial tool coordinate system
      kinPlusKinematics : Bool;   // 4D and lower have an implicit rotation of C = -180°.
      toolFrames : Array[1..3] of "LKinCtrl_typeFrame";   // tool frames
   END_VAR

   VAR_IN_OUT 
      positionInitialAndResult : Array[1..6] of LReal;   // position to be transformed in cartesian CS
   END_VAR

   VAR_TEMP 
      tempPosition : Array[1..6] of LReal;
      tempWcsToTCSInitial : Array[1..3, 1..3] of LReal;
      tempTCSInitialToFCS : Array[1..3, 1..3] of LReal;
      tempFCSToTCSResult : Array[1..3, 1..3] of LReal;
      tempWcsToFCS : Array[1..3, 1..3] of LReal;
      tempWcsToTCSResult : Array[1..3, 1..3] of LReal;
      tempPFCSToTCSResult : Array[1..3, 1..1] of LReal;
      tempPTCSInitialToFCS : Array[1..3, 1..1] of LReal;
      tempPWCSToTCSInitial : Array[1..3, 1..1] of LReal;
      tempPResult : Array[1..3, 1..1] of LReal;
      tempBool : Bool;
      tempWord : Word;
   END_VAR


BEGIN
	//==========================================================================================
	// SIEMENS AG
	// (c)Copyright 2020 All Rights Reserved
	//------------------------------------------------------------------------------------------
	// Library: LKinCtrl
	// Tested with: S7-1517T-3 PN/DP
	// Engineering: TIA Portal V19
	// Restrictions: ---
	// Requirements: S7-1500T FW 3.1
	// Functionality: LKinCtrl_FrameTransTool
	// The FC transforms a given WCS position of a tool into the WCS position of another tool  
	//
	// Support: tech.team.motioncontrol@siemens.com
	// Note: Parameter comments are only available in language 'English (United States)'
	//------------------------------------------------------------------------------------------
	// Change log table:
	// Version    Date          Expert in charge    Changes applied
	// 01.00.00   08.08.2024    JH                  First release version v1.0
	//===========================================================================================
	
	// Check if last CS differs from actual CS
	IF #toolResult = #toolInitial
	  OR #toolInitial < 1 OR #toolInitial > 3
	  OR #toolResult < 1 OR #toolResult > 3
	THEN
	  // No calculation needed --> Return
	  RETURN;
	END_IF;
	
	// WCS is just a placeholder and describes the cartesian coordinate system of the input frame, e.g. OCS 1-3 or UCS
	REGION CREATE_ROTATION_MATRICES
	  // Create rotation matrix WCS in TCS initial
	  // Rxyz(A,B,C) = [Rz(A) * Ry(B) * Rx(C)]
	  "LKinCtrl_RotXYZ"(angleA       := #positionInitialAndResult[4],
	                    angleB       := #positionInitialAndResult[5],
	                    angleC       := SEL(G := #kinPlusKinematics, IN0 := -180, IN1 := #positionInitialAndResult[6]), // implicit rotation of C = -180 for 4D and lower
	                    resultMatrix := #tempWcsToTCSInitial);
	  
	  // Create rotation matrix TCS initial in FCS
	  // Rxyz(A,B,C) = [Rz(A) * Ry(B) * Rx(C)]^T
	  "LKinCtrl_RotXYZTranspose"(angleA       := #toolFrames[#toolInitial].a,
	                             angleB       := #toolFrames[#toolInitial].b,
	                             angleC       := #toolFrames[#toolInitial].c,
	                             resultMatrix := #tempTCSInitialToFCS);
	  
	  // Create rotation matrix FCS in TCS result
	  // Rxyz(A,B,C) = [Rz(A) * Ry(B) * Rx(C)]
	  "LKinCtrl_RotXYZ"(angleA       := #toolFrames[#toolResult].a,
	                    angleB       := #toolFrames[#toolResult].b,
	                    angleC       := #toolFrames[#toolResult].c,
	                    resultMatrix := #tempFCSToTCSResult);
	  
	  // Rotation WCS to FCS
	  "LKinCtrl_MatrixMultiplication"(status       => #tempWord,
	                                  matrix1      := #tempWcsToTCSInitial,
	                                  matrix2      := #tempTCSInitialToFCS,
	                                  matrixResult := #tempWcsToFCS,
	                                  error        => #tempBool);
	  
	  // Rotation WCS to TCS result
	  "LKinCtrl_MatrixMultiplication"(status       => #tempWord,
	                                  matrix1      := #tempWcsToFCS,
	                                  matrix2      := #tempFCSToTCSResult,
	                                  matrixResult := #tempWcsToTCSResult,
	                                  error        => #tempBool);
	END_REGION
	
	REGION TRANSLATION
	  // Translation from TCS initial to FCS (in FCS)
	  #tempPTCSInitialToFCS[1, 1] := - #toolFrames[#toolInitial].x;
	  #tempPTCSInitialToFCS[2, 1] := - #toolFrames[#toolInitial].y;
	  #tempPTCSInitialToFCS[3, 1] := - #toolFrames[#toolInitial].z;
	  // Translation from TCS initial to FCS (in WCS)
	  "LKinCtrl_MatrixMultiplication"(status       => #tempWord,
	                                  matrix1      := #tempWcsToFCS,
	                                  matrix2      := #tempPTCSInitialToFCS,
	                                  matrixResult := #tempPResult,
	                                  error        => #tempBool);
	  #tempPTCSInitialToFCS := #tempPResult;
	  
	  //Translation from FCS to TCS result (in FCS)
	  #tempPFCSToTCSResult[1, 1] := #toolFrames[#toolResult].x;
	  #tempPFCSToTCSResult[2, 1] := #toolFrames[#toolResult].y;
	  #tempPFCSToTCSResult[3, 1] := #toolFrames[#toolResult].z;
	  //Translation from FCS to TCS result (in WCS)
	  "LKinCtrl_MatrixMultiplication"(status       => #tempWord,
	                                  matrix1      := #tempWcsToFCS,
	                                  matrix2      := #tempPFCSToTCSResult,
	                                  matrixResult := #tempPResult,
	                                  error        => #tempBool);
	  #tempPFCSToTCSResult := #tempPResult;
	  
	  //Translation from WCS to TCS initial (in WCS)
	  #tempPWCSToTCSInitial[1, 1] := #positionInitialAndResult[1];
	  #tempPWCSToTCSInitial[2, 1] := #positionInitialAndResult[2];
	  #tempPWCSToTCSInitial[3, 1] := #positionInitialAndResult[3];
	  
	  // translation (all expressed in WCS)
	  #positionInitialAndResult[1] := #tempPWCSToTCSInitial[1, 1] + #tempPTCSInitialToFCS[1, 1] + #tempPFCSToTCSResult[1, 1];
	  #positionInitialAndResult[2] := #tempPWCSToTCSInitial[2, 1] + #tempPTCSInitialToFCS[2, 1] + #tempPFCSToTCSResult[2, 1];
	  #positionInitialAndResult[3] := #tempPWCSToTCSInitial[3, 1] + #tempPTCSInitialToFCS[3, 1] + #tempPFCSToTCSResult[3, 1];
	END_REGION
	
	REGION ROTATION
	  // inverse problem from rotation matrix back to A,B,C
	  "LKinCtrl_InvRotXYZ"(rotMatrix := #tempWcsToTCSResult,
	                       A         => #positionInitialAndResult[4],
	                       B         => #positionInitialAndResult[5],
	                       C         => #positionInitialAndResult[6]);
	  
	  // force b and c to 0 for 4D and lower - also resets implicit rotation of C = -180 for 4D and lower
	  #positionInitialAndResult[5] := SEL(G := #kinPlusKinematics, IN0 := 0, IN1 := #positionInitialAndResult[5]);
	  #positionInitialAndResult[6] := SEL(G := #kinPlusKinematics, IN0 := 0, IN1 := #positionInitialAndResult[6]);
	END_REGION
	
	
END_FUNCTION

DATA_BLOCK "instFB_AutoCtrl_ABCDE"   // DB
TITLE = ABCDE Auto Cycle instance DB
{ S7_Optimized_Access := 'TRUE' }
// iDB for FB_AutoCtrl_ABCDE — Wang Shuo 4-REGION ABCDE 6-state machine + MC_MoveLinearAbsolute
// stored: InstanceOfName FB_AutoCtrl_ABCDE, InstanceOfType FB
"FB_AutoCtrl_ABCDE"
BEGIN
END_DATA_BLOCK

DATA_BLOCK "instFB_AxisCtrl"   // DB
TITLE = Axis Control instance DB
{ S7_Optimized_Access := 'TRUE' }
// iDB for FB_AxisCtrl — per-axis MC_Power/Home/Reset for SCARA 4-joint kinematic
// stored: InstanceOfName FB_AxisCtrl, InstanceOfType FB
"FB_AxisCtrl"
BEGIN
END_DATA_BLOCK

DATA_BLOCK "instFB_MCDDataTransfer"   // DB
TITLE = MCD Data Transfer instance DB
{ S7_Optimized_Access := 'TRUE' }
// iDB for FB_MCDDataTransfer — publishes ScaraArm3D.AxesData.A[i].{Position,Velocity} to GDB_MCDData for NX MCD viewport
// stored: InstanceOfName FB_MCDDataTransfer, InstanceOfType FB
"FB_MCDDataTransfer"
BEGIN
END_DATA_BLOCK

DATA_BLOCK "instFB_AutoCtrl_5Pts"   // DB23
VERSION : 1.1
// Instance DB for FB_AutoCtrl_5Pts (Phase 4a, 2026-05-21). Huashili-pattern CASE auto FB; replaces FB_AutoCtrl_ABCDE. DB number may be auto-assigned by TIA on import.
// stored: InstanceOfName FB_AutoCtrl_5Pts, InstanceOfType FB
"FB_AutoCtrl_5Pts"
BEGIN
END_DATA_BLOCK

DATA_BLOCK "instFB_AutoCtrl_Palletizing"   // DB
TITLE = instFB_AutoCtrl_Palletizing (C69 Phase 2.2)
VERSION : 1.1
// C69 Phase 2.2 (2026-05-18) — instance DB for FB_AutoCtrl_Palletizing. 48-element pts[] holds 16 boxes x 3 phases (approach/place/retract) for the 4-layer stacking pattern. instMoveLinAbs has NO AttributeList so SetPoint defaults to FALSE (required for MC_MoveLinearAbsolute Execute pulse to reach MC subsystem; lesson from Phase G C67 rev 0.1 failure).
// stored: InstanceOfName FB_AutoCtrl_Palletizing, InstanceOfType FB
"FB_AutoCtrl_Palletizing"
BEGIN
END_DATA_BLOCK

DATA_BLOCK "instFB_ConveyorCtrl"   // DB
TITLE = instFB_ConveyorCtrl (infeed modularisation, 2026-05-20)
VERSION : 1.1
// Instance DB for FB_ConveyorCtrl (2026-05-20). Owns the palletizing infeed -- SpawnContainerCmd pulse + BeltVelocity belt latch. No MC instances, so zero OB91 (MC-Servo) impact. DB number omitted -- TIA auto-assigns.
// stored: InstanceOfName FB_ConveyorCtrl, InstanceOfType FB
"FB_ConveyorCtrl"
BEGIN
END_DATA_BLOCK

DATA_BLOCK "instFB_HMIStatusMirror"   // DB14
TITLE = instFB_HMIStatusMirror (Phase 2.4)
VERSION : 1.1
// Phase 2.4 (C71, 2026-05-18) — instance DB for FB_HMIStatusMirror. Pure mirror FB; no statics (only VAR_TEMP for activeMode arbitration). Tiny iDB schema.
// stored: InstanceOfName FB_HMIStatusMirror, InstanceOfType FB
"FB_HMIStatusMirror"
BEGIN
END_DATA_BLOCK

DATA_BLOCK "instFB_Init"   // DB22
VERSION : 1.1
// Instance DB for FB_Init (Phase 3, 2026-05-21). Homing block - LKinCtrl_MC_GroupHome on ScaraArm3D, runs in OB30. DB number may be auto-assigned by TIA on import.
// stored: InstanceOfName FB_Init, InstanceOfType FB
"FB_Init"
BEGIN
END_DATA_BLOCK

DATA_BLOCK "instFB_ManualCtrl"   // DB
TITLE = instFB_ManualCtrl (Phase G)
VERSION : 1.1
// Phase G (C67, 2026-05-18) — instance DB for FB_ManualCtrl. Holds 4 MC_MoveJog + 1 MC_MoveLinearAbsolute + 1 R_TRIG + 1 Bool static. Total 6 multi-instance MC slots; with FB_AxisCtrl's 14 + FB_AutoCtrl_ABCDE's 1 = 21 declared system-wide, well under OB91 budget.
// stored: InstanceOfName FB_ManualCtrl, InstanceOfType FB
"FB_ManualCtrl"
BEGIN
END_DATA_BLOCK

DATA_BLOCK "instFB_PatternAutoGen"   // DB25
VERSION : 1.1
// stored: InstanceOfName FB_PatternAutoGen, InstanceOfType FB
"FB_PatternAutoGen"
BEGIN
END_DATA_BLOCK

DATA_BLOCK "instFB_TeachCtrl"   // DB28
VERSION : 1.1
// Instance DB for FB_TeachCtrl V1.0 (Module F, 2026-05-23). 7 R_TRIG edge detectors (Capture, Verify, Clear, ClearAll, StartReplay, StopReplay, MoveDone) + statTeachOK gate. FB writes to shared GDB_AxisCtrl.LKinCtrl.input.{jogframe, movelinear} - no local MC instance.
// stored: InstanceOfName FB_TeachCtrl, InstanceOfType FB
"FB_TeachCtrl"
BEGIN
END_DATA_BLOCK

DATA_BLOCK "ScaraArm3D"   // DB17, Motion_DB
// stored: InstanceOfName TO_Kinematics, OfSystemLibElement TO_Kinematics, OfSystemLibVersion 9.0
TO_Kinematics   // technology object, version 9.0
   // // inherited from TO_Object
   // VAR
   //    Tcp { ExternalWritable := 'False'; S7_SetPoint := 'True'} : TO_Struct_Kinematics_StatusKinematicsFrameTcp;
   //    Kinematics { S7_SetPoint := 'True'} : TO_Struct_Kinematics_Kinematics;
   //    KcsFrame { S7_SetPoint := 'True'} : TO_Struct_Kinematics_Frame;
   //    OcsFrame { S7_SetPoint := 'True'} : Array[1..3] of TO_Struct_Kinematics_Frame;
   //    Tool { S7_SetPoint := 'True'} : Array[1..3] of TO_Struct_Kinematics_Tool;
   //    DynamicDefaults { S7_SetPoint := 'True'} : TO_Struct_Kinematics_DynamicDefaults;
   //    DynamicLimits { S7_SetPoint := 'True'} : TO_Struct_Kinematics_DynamicLimits;
   //    Joint { S7_SetPoint := 'True'} : TO_Struct_Kinematics_Joint;
   //    AxisCoupling { S7_SetPoint := 'True'} : TO_Struct_Kinematics_AxisCoupling;
   //    MotionQueue { ExternalWritable := 'False'; S7_SetPoint := 'True'} : TO_Struct_Kinematics_MotionQueue;
   //    Transition { S7_SetPoint := 'True'} : TO_Struct_Kinematics_Transition;
   //    Override { S7_SetPoint := 'True'} : TO_Struct_Kinematics_Override;
   //    Conveyor { S7_SetPoint := 'True'} : TO_Struct_Kinematics_Conveyor;
   //    WorkspaceZone { S7_SetPoint := 'True'} : Array[1..10] of TO_Struct_Kinematics_WorkSpaceZone;
   //    KinematicsZone { S7_SetPoint := 'True'} : Array[2..10] of TO_Struct_Kinematics_KinematicsZone;
   //    StatusPath { ExternalWritable := 'False'; S7_SetPoint := 'True'} : TO_Struct_Kinematics_StatusPath;
   //    TcpInWcs { ExternalWritable := 'False'; S7_SetPoint := 'True'} : TO_Struct_Kinematics_StatusKinematicsFrameWithDynamics;
   //    TcpInOcs { ExternalWritable := 'False'; S7_SetPoint := 'True'} : Array[1..3] of TO_Struct_Kinematics_StatusKinematicsFrameWithDynamicsOcs;
   //    StatusOcsFrame { ExternalWritable := 'False'; S7_SetPoint := 'True'} : Array[1..3] of TO_Struct_Kinematics_StatusFrame;
   //    StatusKinematics { ExternalWritable := 'False'; S7_SetPoint := 'True'} : TO_Struct_Kinematics_StatusKinematics;
   //    AxesData { ExternalWritable := 'False'; S7_SetPoint := 'True'} : TO_Struct_Kinematics_AxesData;
   //    JointData { ExternalWritable := 'False'; S7_SetPoint := 'True'} : TO_Struct_Kinematics_StatusJointData;
   //    FlangeInKcs { ExternalWritable := 'False'; S7_SetPoint := 'True'} : TO_Struct_Kinematics_StatusFlangeInKcs;
   //    StatusTool { ExternalWritable := 'False'; S7_SetPoint := 'True'} : TO_Struct_Kinematics_StatusTool;
   //    StatusConveyor { ExternalWritable := 'False'; S7_SetPoint := 'True'} : Array[1..3] of TO_Struct_Kinematics_StatusConveyor;
   //    StatusWorkspaceZone { ExternalWritable := 'False'; S7_SetPoint := 'True'} : Array[1..10] of TO_Struct_Kinematics_StatusWorkSpaceZone;
   //    StatusKinematicsZone { ExternalWritable := 'False'; S7_SetPoint := 'True'} : Array[2..10] of TO_Struct_Kinematics_StatusKinematicsZone;
   //    StatusZoneMonitoring { ExternalWritable := 'False'; S7_SetPoint := 'True'} : TO_Struct_Kinematics_StatusZoneMonitoring;
   //    StatusMotionQueue { ExternalWritable := 'False'; S7_SetPoint := 'True'} : TO_Struct_Kinematics_StatusMotionQueue;
   //    KinematicsAxis { ExternalWritable := 'False'; S7_SetPoint := 'True'} : TO_Struct_Kinematics_KinematicsAxis;
   //    Units { ExternalWritable := 'False'; S7_SetPoint := 'True'} : TO_Struct_Kinematics_Units;
   //    StatusInterpreterMotion { ExternalWritable := 'False'; S7_SetPoint := 'True'} : TO_Struct_Kinematics_StatusInterpreterMotion;
   //    StatusWord { ExternalWritable := 'False'} : DWord;
   //    ErrorWord { ExternalWritable := 'False'} : DWord;
   //    ErrorDetail { ExternalWritable := 'False'; S7_SetPoint := 'True'} : TO_Struct_ErrorDetail;
   //    WarningWord { ExternalWritable := 'False'} : DWord;
   //    ControlPanel { S7_SetPoint := 'True'} : TO_Struct_Kinematics_ControlPanel;
   //    InternalToTrace { S7_SetPoint := 'True'} : Array[1..4] of TO_Struct_Internal;
   // END_VAR
BEGIN
   Kinematics.TypeOfKinematics := 10;
   Kinematics.Parameter[2] := 1150.0;
   Kinematics.Parameter[5] := 1200.0;
   Kinematics.Parameter[9..32] := 0.0;
   KcsFrame.x := 0.0;
   KcsFrame.y := 0.0;
   KcsFrame.z := 0.0;
   KcsFrame."a" := 0.0;
   KcsFrame."b" := 0.0;
   KcsFrame.c := 0.0;
   OcsFrame[2..3].x := 0.0;
   OcsFrame[2..3].y := 0.0;
   OcsFrame[2..3].z := 0.0;
   OcsFrame[2..3]."a" := 0.0;
   OcsFrame[1..3]."b" := 0.0;
   OcsFrame[1..3].c := 0.0;
   Tool[2..3].Frame.x := 0.0;
   Tool[2..3].Frame.y := 0.0;
   Tool[1].Frame.z := 50.0;
   Tool[2..3].Frame.z := 0.0;
   Tool[1..3].Frame."a" := 0.0;
   DynamicDefaults.Path.Velocity := 2000.0;
   DynamicDefaults.Path.Acceleration := 10000.0;
   DynamicDefaults.Path.Deceleration := 10000.0;
   DynamicDefaults.Path.Jerk := 100000.0;
   DynamicDefaults.Orientation.Velocity := 2000.0;
   DynamicDefaults.Orientation.Acceleration := 20000.0;
   DynamicDefaults.Orientation.Deceleration := 20000.0;
   DynamicDefaults.Orientation.Jerk := 1000000.0;
   DynamicDefaults.DynamicAdaption := 1;
   DynamicDefaults.MoveDirect.VelocityFactor := 0.5;
   DynamicDefaults.MoveDirect.AccelerationFactor := 0.5;
   DynamicDefaults.MoveDirect.DecelerationFactor := 0.5;
   DynamicDefaults.MoveDirect.JerkFactor := 0.5;
   DynamicLimits.Path.Velocity := 3000.0;
   DynamicLimits.Path.Acceleration := 100000.0;
   DynamicLimits.Path.Deceleration := 100000.0;
   DynamicLimits.Orientation.Velocity := 2200.0;
   DynamicLimits.Orientation.Acceleration := 20000.0;
   DynamicLimits.Orientation.Deceleration := 20000.0;
   DynamicLimits.Orientation.Jerk := 1000000.0;
   Override.Velocity := 62.0;
   WorkspaceZone[1].Active := true;
   WorkspaceZone[2..10].Active := false;
   WorkspaceZone[1].Valid := true;
   WorkspaceZone[2..10].Valid := false;
   WorkspaceZone[2..10]."Type" := 1;
   WorkspaceZone[1..10].ReferenceSystem := 0;
   WorkspaceZone[2..10].Frame.x := 0.0;
   WorkspaceZone[2..10].Frame.y := 0.0;
   WorkspaceZone[1].Frame.z := -100.0;
   WorkspaceZone[2..10].Frame.z := 0.0;
   WorkspaceZone[1..10].Frame."a" := 0.0;
   WorkspaceZone[1..10].Frame."b" := 0.0;
   WorkspaceZone[1..10].Frame.c := 0.0;
   WorkspaceZone[1].Geometry."Type" := 2;
   WorkspaceZone[2..10].Geometry."Type" := 0;
   WorkspaceZone[1].Geometry.Parameter[1] := 2500.0;
   WorkspaceZone[1].Geometry.Parameter[2] := 2000.0;
   WorkspaceZone[1].Geometry.Parameter[3] := 500.0;
   WorkspaceZone[2].Geometry.Parameter[1..3] := 500.0;
   WorkspaceZone[3].Geometry.Parameter[1..3] := 500.0;
   WorkspaceZone[4].Geometry.Parameter[1..3] := 500.0;
   WorkspaceZone[5].Geometry.Parameter[1..3] := 500.0;
   WorkspaceZone[6].Geometry.Parameter[1..3] := 500.0;
   WorkspaceZone[7].Geometry.Parameter[1..3] := 500.0;
   WorkspaceZone[8].Geometry.Parameter[1..3] := 500.0;
   WorkspaceZone[9].Geometry.Parameter[1..3] := 500.0;
   WorkspaceZone[10].Geometry.Parameter[1..3] := 500.0;
   KinematicsZone[3..10].Active := false;
   KinematicsZone[3..10].Valid := false;
   KinematicsZone[2..10].ReferenceSystem := 0;
   KinematicsZone[2..10].Frame.x := 0.0;
   KinematicsZone[2..10].Frame.y := 0.0;
   KinematicsZone[2..10].Frame.z := 0.0;
   KinematicsZone[2..10].Frame."a" := 0.0;
   KinematicsZone[2..10].Frame."b" := 0.0;
   KinematicsZone[2..10].Frame.c := 0.0;
   KinematicsZone[2].Geometry."Type" := 2;
   KinematicsZone[3..10].Geometry."Type" := 0;
   KinematicsZone[2].Geometry.Parameter[1] := 5000.0;
   KinematicsZone[2].Geometry.Parameter[2] := 3000.0;
   KinematicsZone[2].Geometry.Parameter[3] := 5000.0;
   KinematicsZone[3].Geometry.Parameter[1..3] := 500.0;
   KinematicsZone[4].Geometry.Parameter[1..3] := 500.0;
   KinematicsZone[5].Geometry.Parameter[1..3] := 500.0;
   KinematicsZone[6].Geometry.Parameter[1..3] := 500.0;
   KinematicsZone[7].Geometry.Parameter[1..3] := 500.0;
   KinematicsZone[8].Geometry.Parameter[1..3] := 500.0;
   KinematicsZone[9].Geometry.Parameter[1..3] := 500.0;
   KinematicsZone[10].Geometry.Parameter[1..3] := 500.0;
   ControlPanel.Input.TimeOut := 2000.0;
   ControlPanel.Input.EsLifeSign := 0;
   ControlPanel.Input.Command[1..2].ReqCounter := 0;
   ControlPanel.Input.Command[1..2]."Type" := 0;
   ControlPanel.Input.Command[1].Position[1..4] := 0.0;
   ControlPanel.Input.Command[2].Position[1..4] := 0.0;
   ControlPanel.Input.Command[1].Velocity[1..2] := 0.0;
   ControlPanel.Input.Command[2].Velocity[1..2] := 0.0;
   ControlPanel.Input.Command[1].Acceleration[1..2] := 0.0;
   ControlPanel.Input.Command[2].Acceleration[1..2] := 0.0;
   ControlPanel.Input.Command[1].Deceleration[1..2] := 0.0;
   ControlPanel.Input.Command[2].Deceleration[1..2] := 0.0;
   ControlPanel.Input.Command[1].Jerk[1..2] := 0.0;
   ControlPanel.Input.Command[2].Jerk[1..2] := 0.0;
   ControlPanel.Input.Command[1].Param[1..9] := 0.0;
   ControlPanel.Input.Command[2].Param[1..9] := 0.0;
   ControlPanel.Input.Command[1..2].CoordinateSystem := 0;
   ControlPanel.Input.Command[1..2].ToolNumber := 0;
   InternalToTrace[1..4].Id := 0;
   InternalToTrace[1..4].Value := 0.0;
   Kinematics.TypeOfKinematics := 10;
END_DATA_BLOCK

